C03651=1200.796,212.274,-59.248,-177.519,6.536,148.464
C03652=1200.800,212.025,-59.224,-177.522,6.534,148.465
C03653=1200.805,211.777,-59.199,-177.524,6.533,148.465
C03654=1200.809,211.528,-59.175,-177.527,6.531,148.466
C03655=1200.814,211.257,-59.148,-177.530,6.528,148.466
C03656=1200.819,210.986,-59.122,-177.533,6.526,148.466
C03657=1200.824,210.716,-59.095,-177.535,6.524,148.466
C03658=1200.829,210.446,-59.069,-177.539,6.522,148.467
C03659=1200.833,210.197,-59.044,-177.541,6.520,148.467
C03660=1200.838,209.949,-59.020,-177.543,6.518,148.467
C03661=1200.843,209.700,-58.995,-177.546,6.516,148.468
C03662=1200.847,209.451,-58.971,-177.549,6.514,148.468
C03663=1200.851,209.202,-58.947,-177.551,6.512,148.468
C03664=1200.856,208.953,-58.923,-177.554,6.510,148.469
C03665=1200.861,208.705,-58.899,-177.557,6.509,148.469
C03666=1200.865,208.456,-58.874,-177.559,6.506,148.469
C03667=1200.870,208.207,-58.849,-177.562,6.505,148.469
C03668=1200.874,207.958,-58.825,-177.565,6.502,148.470
C03669=1200.879,207.710,-58.801,-177.567,6.500,148.470
C03670=1200.884,207.461,-58.777,-177.570,6.498,148.470
C03671=1200.888,207.212,-58.753,-177.573,6.497,148.471
C03672=1200.893,206.963,-58.728,-177.575,6.495,148.471
C03673=1200.897,206.714,-58.704,-177.578,6.493,148.471
C03674=1200.902,206.466,-58.680,-177.580,6.491,148.472
C03675=1200.906,206.217,-58.657,-177.583,6.489,148.472
C03676=1200.912,205.968,-58.632,-177.585,6.487,148.472
C03677=1200.915,205.719,-58.608,-177.588,6.485,148.473
C03678=1200.920,205.471,-58.584,-177.591,6.483,148.473
C03679=1200.925,205.221,-58.560,-177.593,6.482,148.473
C03680=1200.930,204.973,-58.536,-177.596,6.480,148.474
C03681=1200.934,204.724,-58.511,-177.598,6.478,148.474
C03682=1200.938,204.475,-58.487,-177.601,6.476,148.474
C03683=1200.943,204.226,-58.463,-177.604,6.474,148.474
C03684=1200.948,203.978,-58.439,-177.606,6.472,148.475
C03685=1200.952,203.729,-58.415,-177.609,6.470,148.475
C03686=1200.957,203.480,-58.392,-177.612,6.468,148.475
C03687=1200.961,203.232,-58.367,-177.615,6.466,148.476
C03688=1200.966,202.982,-58.344,-177.617,6.464,148.476
C03689=1200.970,202.733,-58.319,-177.620,6.462,148.476
C03690=1200.975,202.485,-58.295,-177.622,6.460,148.476
C03691=1200.979,202.236,-58.272,-177.625,6.458,148.477
C03692=1200.984,201.987,-58.248,-177.627,6.456,148.477
C03693=1200.988,201.738,-58.224,-177.630,6.455,148.478
C03694=1200.994,201.490,-58.200,-177.633,6.453,148.478
C03695=1200.998,201.241,-58.176,-177.635,6.451,148.478
C03696=1201.003,200.992,-58.152,-177.638,6.449,148.479
C03697=1201.006,200.743,-58.128,-177.641,6.447,148.479
C03698=1201.011,200.494,-58.104,-177.643,6.446,148.479
C03699=1201.016,200.246,-58.080,-177.646,6.444,148.480
C03700=1201.020,199.997,-58.057,-177.649,6.442,148.480
C03701=1201.025,199.748,-58.033,-177.651,6.440,148.480
C03702=1201.029,199.499,-58.009,-177.654,6.438,148.480
C03703=1201.035,199.250,-57.985,-177.656,6.436,148.481
C03704=1201.039,199.001,-57.961,-177.659,6.434,148.481
C03705=1201.044,198.752,-57.938,-177.661,6.433,148.481
C03706=1201.048,198.504,-57.914,-177.664,6.431,148.482
C03707=1201.053,198.255,-57.891,-177.667,6.429,148.482
C03708=1201.057,198.007,-57.867,-177.669,6.427,148.482
C03709=1201.062,197.758,-57.843,-177.672,6.425,148.483
C03710=1201.067,197.508,-57.820,-177.675,6.423,148.483
C03711=1201.071,197.260,-57.796,-177.677,6.422,148.484
C03712=1201.076,197.011,-57.772,-177.680,6.420,148.484
C03713=1201.080,196.761,-57.749,-177.683,6.418,148.484
C03714=1201.084,196.513,-57.725,-177.685,6.416,148.485
C03715=1201.089,196.264,-57.701,-177.688,6.414,148.485
C03716=1201.094,196.015,-57.678,-177.690,6.412,148.485
C03717=1201.098,195.766,-57.654,-177.693,6.410,148.485
C03718=1201.103,195.517,-57.630,-177.696,6.409,148.486
C03719=1201.108,195.268,-57.607,-177.698,6.407,148.486
C03720=1201.112,195.019,-57.584,-177.701,6.405,148.486
C03721=1201.117,194.771,-57.560,-177.703,6.403,148.487
C03722=1201.121,194.522,-57.536,-177.706,6.401,148.487
C03723=1201.127,194.274,-57.513,-177.709,6.399,148.487
C03724=1201.131,194.025,-57.490,-177.711,6.398,148.488
C03725=1201.136,193.776,-57.466,-177.714,6.396,148.488
C03726=1201.140,193.527,-57.443,-177.717,6.394,148.488
C03727=1201.144,193.278,-57.420,-177.719,6.392,148.489
C03728=1201.149,193.029,-57.396,-177.722,6.390,148.489
C03729=1201.154,192.780,-57.373,-177.725,6.389,148.490
C03730=1201.159,192.531,-57.350,-177.727,6.387,148.490
C03731=1201.163,192.283,-57.326,-177.730,6.385,148.490
C03732=1201.168,192.034,-57.302,-177.733,6.383,148.491
C03733=1201.172,191.785,-57.279,-177.735,6.381,148.491
C03734=1201.177,191.536,-57.256,-177.738,6.380,148.491
C03735=1201.181,191.287,-57.233,-177.741,6.378,148.492
C03736=1201.186,191.038,-57.209,-177.743,6.376,148.492
C03737=1201.190,190.789,-57.186,-177.746,6.374,148.492
C03738=1201.195,190.540,-57.163,-177.748,6.373,148.493
C03739=1201.200,190.292,-57.140,-177.751,6.371,148.493
C03740=1201.205,190.043,-57.116,-177.753,6.369,148.493
C03741=1201.209,189.794,-57.094,-177.756,6.368,148.494
C03742=1201.214,189.545,-57.070,-177.758,6.366,148.494
C03743=1201.218,189.296,-57.047,-177.761,6.364,148.494
C03744=1201.223,189.047,-57.023,-177.764,6.362,148.495
C03745=1201.228,188.798,-57.000,-177.766,6.360,148.495
C03746=1201.232,188.549,-56.977,-177.769,6.358,148.495
C03747=1201.237,188.301,-56.954,-177.772,6.356,148.496
C03748=1201.242,188.052,-56.931,-177.774,6.355,148.496
C03749=1201.247,187.803,-56.908,-177.777,6.353,148.496
C03750=1201.250,187.554,-56.885,-177.779,6.351,148.497
C03751=1201.255,187.305,-56.862,-177.782,6.349,148.497
C03752=1201.260,187.056,-56.838,-177.785,6.347,148.497
C03753=1201.265,186.807,-56.815,-177.787,6.346,148.498
C03754=1201.269,186.559,-56.792,-177.790,6.344,148.498
C03755=1201.274,186.310,-56.769,-177.792,6.343,148.499
C03756=1201.279,186.061,-56.746,-177.795,6.341,148.499
C03757=1201.282,185.812,-56.723,-177.798,6.339,148.499
C03758=1201.288,185.562,-56.700,-177.801,6.338,148.500
C03759=1201.293,185.293,-56.675,-177.803,6.336,148.500
C03760=1201.297,185.024,-56.650,-177.807,6.333,148.500
C03761=1201.302,184.754,-56.625,-177.809,6.331,148.501
C03762=1201.308,184.484,-56.600,-177.812,6.330,148.501
C03763=1201.312,184.235,-56.577,-177.815,6.328,148.502
C03764=1201.317,183.987,-56.555,-177.817,6.326,148.502
C03765=1201.321,183.738,-56.532,-177.820,6.324,148.502
C03766=1201.326,183.489,-56.509,-177.822,6.323,148.503
C03767=1201.331,183.240,-56.486,-177.825,6.321,148.503
C03768=1201.336,182.991,-56.464,-177.827,6.320,148.503
C03769=1201.340,182.742,-56.440,-177.830,6.318,148.504
C03770=1201.344,182.493,-56.418,-177.833,6.316,148.504
C03771=1201.349,182.244,-56.395,-177.836,6.315,148.505
C03772=1201.354,181.995,-56.372,-177.838,6.313,148.505
C03773=1201.358,181.747,-56.349,-177.841,6.311,148.505
C03774=1201.363,181.498,-56.326,-177.844,6.309,148.506
C03775=1201.367,181.248,-56.304,-177.846,6.307,148.506
C03776=1201.372,180.999,-56.281,-177.848,6.306,148.506
C03777=1201.377,180.751,-56.259,-177.851,6.305,148.507
C03778=1201.382,180.502,-56.235,-177.854,6.303,148.507
C03779=1201.386,180.253,-56.213,-177.856,6.301,148.507
C03780=1201.391,180.004,-56.190,-177.859,6.299,148.508
C03781=1201.395,179.755,-56.168,-177.862,6.297,148.508
C03782=1201.400,179.506,-56.144,-177.864,6.296,148.509
C03783=1201.404,179.257,-56.122,-177.867,6.294,148.509
C03784=1201.410,179.008,-56.099,-177.870,6.292,148.509
C03785=1201.414,178.759,-56.077,-177.872,6.291,148.510
C03786=1201.418,178.510,-56.054,-177.875,6.289,148.510
C03787=1201.423,178.261,-56.032,-177.877,6.287,148.510
C03788=1201.428,178.012,-56.009,-177.880,6.286,148.511
C03789=1201.432,177.763,-55.987,-177.883,6.284,148.511
C03790=1201.438,177.515,-55.964,-177.886,6.282,148.512
C03791=1201.442,177.265,-55.942,-177.888,6.280,148.512
C03792=1201.447,177.016,-55.918,-177.890,6.279,148.512
C03793=1201.451,176.768,-55.897,-177.893,6.278,148.513
C03794=1201.455,176.519,-55.874,-177.896,6.276,148.513
C03795=1201.460,176.269,-55.851,-177.898,6.274,148.514
C03796=1201.465,176.021,-55.829,-177.901,6.272,148.514
C03797=1201.470,175.772,-55.806,-177.904,6.270,148.514
C03798=1201.474,175.522,-55.784,-177.906,6.269,148.515
C03799=1201.479,175.274,-55.762,-177.909,6.268,148.515
C03800=1201.484,175.025,-55.739,-177.911,6.266,148.515
C03801=1201.488,174.777,-55.717,-177.914,6.264,148.516
C03802=1201.493,174.527,-55.695,-177.917,6.262,148.516
C03803=1201.498,174.278,-55.672,-177.920,6.261,148.517
C03804=1201.502,174.030,-55.650,-177.922,6.259,148.517
C03805=1201.506,173.780,-55.628,-177.925,6.257,148.517
C03806=1201.512,173.531,-55.605,-177.927,6.256,148.518
C03807=1201.516,173.283,-55.583,-177.930,6.254,148.518
C03808=1201.520,173.033,-55.561,-177.932,6.253,148.518
C03809=1201.526,172.784,-55.538,-177.935,6.251,148.519
C03810=1201.530,172.536,-55.515,-177.938,6.249,148.519
C03811=1201.535,172.287,-55.494,-177.940,6.247,148.520
C03812=1201.540,172.037,-55.471,-177.943,6.246,148.520
C03813=1201.545,171.789,-55.449,-177.946,6.245,148.521
C03814=1201.549,171.540,-55.427,-177.948,6.243,148.521
C03815=1201.554,171.290,-55.404,-177.951,6.241,148.521
C03816=1201.558,171.042,-55.382,-177.954,6.239,148.522
C03817=1201.563,170.792,-55.360,-177.956,6.238,148.522
C03818=1201.567,170.544,-55.338,-177.958,6.237,148.522
C03819=1201.572,170.295,-55.315,-177.961,6.235,148.523
C03820=1201.577,170.046,-55.294,-177.964,6.233,148.523
C03821=1201.581,169.797,-55.272,-177.966,6.231,148.523
C03822=1201.586,169.548,-55.250,-177.970,6.230,148.524
C03823=1201.591,169.299,-55.228,-177.972,6.229,148.524
C03824=1201.596,169.050,-55.205,-177.974,6.227,148.525
C03825=1201.600,168.801,-55.183,-177.977,6.225,148.525
C03826=1201.605,168.552,-55.161,-177.980,6.223,148.526
C03827=1201.609,168.303,-55.139,-177.982,6.222,148.526
C03828=1201.614,168.054,-55.117,-177.985,6.221,148.526
C03829=1201.619,167.805,-55.095,-177.987,6.219,148.527
C03830=1201.624,167.556,-55.073,-177.990,6.217,148.527
C03831=1201.628,167.307,-55.051,-177.993,6.216,148.528
C03832=1201.633,167.058,-55.029,-177.996,6.214,148.528
C03833=1201.637,166.809,-55.007,-177.998,6.213,148.528
C03834=1201.642,166.560,-54.986,-178.000,6.211,148.529
C03835=1201.647,166.311,-54.964,-178.003,6.209,148.529
C03836=1201.652,166.062,-54.941,-178.006,6.207,148.529
C03837=1201.656,165.812,-54.919,-178.009,6.206,148.530
C03838=1201.661,165.564,-54.898,-178.011,6.205,148.530
C03839=1201.666,165.315,-54.876,-178.014,6.203,148.531
C03840=1201.670,165.066,-54.854,-178.016,6.201,148.531
C03841=1201.675,164.817,-54.832,-178.019,6.200,148.532
C03842=1201.680,164.568,-54.810,-178.022,6.198,148.532
C03843=1201.684,164.319,-54.788,-178.024,6.197,148.532
C03844=1201.689,164.070,-54.766,-178.027,6.195,148.533
C03845=1201.694,163.821,-54.745,-178.030,6.194,148.533
C03846=1201.698,163.572,-54.723,-178.032,6.192,148.534
C03847=1201.703,163.323,-54.701,-178.034,6.191,148.534
C03848=1201.708,163.075,-54.679,-178.037,6.189,148.534
C03849=1201.712,162.825,-54.657,-178.040,6.187,148.535
C03850=1201.717,162.577,-54.636,-178.043,6.186,148.535
C03851=1201.721,162.327,-54.614,-178.045,6.185,148.536
C03852=1201.726,162.078,-54.593,-178.048,6.183,148.536
C03853=1201.731,161.829,-54.571,-178.050,6.181,148.536
C03854=1201.735,161.580,-54.549,-178.053,6.179,148.537
C03855=1201.740,161.331,-54.527,-178.056,6.178,148.537
C03856=1201.744,161.082,-54.505,-178.058,6.177,148.538
C03857=1201.750,160.833,-54.484,-178.061,6.175,148.538
C03858=1201.755,160.584,-54.462,-178.064,6.173,148.539
C03859=1201.759,160.335,-54.440,-178.066,6.172,148.539
C03860=1201.764,160.086,-54.419,-178.068,6.171,148.539
C03861=1201.769,159.837,-54.398,-178.071,6.169,148.540
C03862=1201.773,159.588,-54.376,-178.074,6.167,148.540
C03863=1201.779,159.318,-54.352,-178.077,6.166,148.541
C03864=1201.783,159.050,-54.329,-178.080,6.164,148.541
C03865=1201.788,158.780,-54.305,-178.083,6.162,148.542
C03866=1201.793,158.511,-54.283,-178.085,6.161,148.542
C03867=1201.798,158.263,-54.261,-178.088,6.160,148.542
C03868=1201.803,158.014,-54.239,-178.091,6.158,148.543
C03869=1201.808,157.764,-54.218,-178.093,6.156,148.543
C03870=1201.812,157.516,-54.196,-178.096,6.155,148.544
C03871=1201.817,157.267,-54.175,-178.098,6.154,148.544
C03872=1201.821,157.017,-54.154,-178.101,6.152,148.544
C03873=1201.826,156.769,-54.132,-178.104,6.150,148.545
C03874=1201.831,156.520,-54.111,-178.107,6.149,148.545
C03875=1201.836,156.271,-54.090,-178.109,6.148,148.546
C03876=1201.840,156.021,-54.068,-178.111,6.146,148.546
C03877=1201.845,155.772,-54.047,-178.114,6.144,148.547
C03878=1201.850,155.524,-54.025,-178.117,6.143,148.547
C03879=1201.855,155.275,-54.005,-178.119,6.142,148.548
C03880=1201.859,155.025,-53.982,-178.122,6.140,148.548
C03881=1201.864,154.777,-53.961,-178.125,6.138,148.548
C03882=1201.869,154.527,-53.940,-178.127,6.137,148.549
C03883=1201.873,154.278,-53.918,-178.130,6.136,148.549
C03884=1201.878,154.029,-53.897,-178.133,6.134,148.550
C03885=1201.883,153.780,-53.876,-178.135,6.133,148.550
C03886=1201.888,153.531,-53.855,-178.137,6.131,148.550
C03887=1201.893,153.282,-53.833,-178.140,6.129,148.551
C03888=1201.897,153.033,-53.812,-178.143,6.128,148.551
C03889=1201.902,152.784,-53.791,-178.145,6.127,148.552
C03890=1201.907,152.535,-53.770,-178.148,6.125,148.552
C03891=1201.911,152.286,-53.749,-178.151,6.123,148.553
C03892=1201.915,152.037,-53.727,-178.153,6.123,148.553
C03893=1201.920,151.787,-53.706,-178.156,6.121,148.554
C03894=1201.925,151.539,-53.685,-178.159,6.119,148.554
C03895=1201.930,151.290,-53.664,-178.161,6.118,148.554
C03896=1201.935,151.041,-53.643,-178.164,6.117,148.555
C03897=1201.939,150.791,-53.621,-178.167,6.115,148.555
C03898=1201.944,150.542,-53.601,-178.169,6.113,148.556
C03899=1201.949,150.293,-53.580,-178.171,6.112,148.556
C03900=1201.954,150.044,-53.558,-178.175,6.111,148.557
C03901=1201.958,149.795,-53.538,-178.177,6.109,148.557
C03902=1201.963,149.546,-53.517,-178.179,6.108,148.557
C03903=1201.968,149.297,-53.495,-178.182,6.106,148.558
C03904=1201.972,149.048,-53.474,-178.185,6.105,148.558
C03905=1201.977,148.799,-53.453,-178.187,6.104,148.559
C03906=1201.982,148.550,-53.432,-178.190,6.102,148.559
C03907=1201.987,148.301,-53.411,-178.193,6.100,148.560
C03908=1201.992,148.052,-53.390,-178.195,6.100,148.560
C03909=1201.996,147.803,-53.370,-178.198,6.098,148.561
C03910=1202.000,147.553,-53.348,-178.201,6.096,148.561
C03911=1202.006,147.304,-53.327,-178.203,6.095,148.561
C03912=1202.010,147.055,-53.307,-178.206,6.094,148.562
C03913=1202.015,146.806,-53.286,-178.209,6.092,148.562
C03914=1202.019,146.558,-53.265,-178.211,6.091,148.563
C03915=1202.024,146.308,-53.244,-178.213,6.089,148.563
C03916=1202.029,146.059,-53.223,-178.217,6.088,148.564
C03917=1202.034,145.810,-53.202,-178.219,6.087,148.564
C03918=1202.039,145.560,-53.181,-178.221,6.085,148.565
C03919=1202.043,145.311,-53.161,-178.224,6.083,148.565
C03920=1202.048,145.063,-53.139,-178.227,6.082,148.566
C03921=1202.052,144.814,-53.119,-178.229,6.081,148.566
C03922=1202.058,144.564,-53.098,-178.232,6.079,148.566
C03923=1202.062,144.315,-53.077,-178.235,6.078,148.567
C03924=1202.067,144.066,-53.056,-178.237,6.076,148.567
C03925=1202.072,143.817,-53.036,-178.240,6.075,148.568
C03926=1202.077,143.568,-53.015,-178.242,6.074,148.568
C03927=1202.081,143.319,-52.995,-178.245,6.072,148.569
C03928=1202.086,143.070,-52.974,-178.247,6.071,148.569
C03929=1202.091,142.821,-52.953,-178.250,6.070,148.569
C03930=1202.095,142.572,-52.933,-178.253,6.068,148.570
C03931=1202.100,142.323,-52.912,-178.255,6.067,148.570
C03932=1202.105,142.074,-52.891,-178.258,6.065,148.571
C03933=1202.109,141.824,-52.869,-178.261,6.064,148.571
C03934=1202.114,141.575,-52.849,-178.263,6.063,148.572
C03935=1202.119,141.326,-52.828,-178.266,6.061,148.572
C03936=1202.124,141.077,-52.808,-178.269,6.059,148.573
C03937=1202.128,140.828,-52.788,-178.271,6.059,148.573
C03938=1202.133,140.578,-52.767,-178.274,6.057,148.574
C03939=1202.138,140.329,-52.747,-178.276,6.056,148.574
C03940=1202.143,140.080,-52.726,-178.279,6.055,148.575
C03941=1202.147,139.831,-52.705,-178.282,6.053,148.575
C03942=1202.152,139.582,-52.685,-178.284,6.052,148.575
C03943=1202.157,139.333,-52.664,-178.287,6.050,148.576
C03944=1202.161,139.084,-52.644,-178.289,6.050,148.576
C03945=1202.166,138.835,-52.623,-178.292,6.048,148.577
C03946=1202.171,138.586,-52.602,-178.295,6.046,148.577
C03947=1202.175,138.337,-52.582,-178.297,6.045,148.578
C03948=1202.180,138.087,-52.562,-178.300,6.044,148.578
C03949=1202.186,137.839,-52.542,-178.303,6.042,148.579
C03950=1202.190,137.590,-52.521,-178.305,6.041,148.579
C03951=1202.195,137.341,-52.501,-178.308,6.039,148.580
C03952=1202.200,137.092,-52.480,-178.310,6.038,148.580
C03953=1202.204,136.843,-52.460,-178.313,6.037,148.581
C03954=1202.209,136.593,-52.440,-178.316,6.035,148.581
C03955=1202.214,136.344,-52.419,-178.318,6.034,148.581
C03956=1202.219,136.095,-52.399,-178.321,6.033,148.582
C03957=1202.223,135.846,-52.378,-178.323,6.032,148.582
C03958=1202.228,135.596,-52.359,-178.326,6.030,148.583
C03959=1202.233,135.347,-52.338,-178.329,6.029,148.583
C03960=1202.237,135.098,-52.317,-178.331,6.028,148.584
C03961=1202.242,134.849,-52.297,-178.334,6.026,148.584
C03962=1202.247,134.600,-52.277,-178.337,6.025,148.585
C03963=1202.252,134.351,-52.257,-178.339,6.024,148.585
C03964=1202.257,134.102,-52.236,-178.341,6.023,148.586
C03965=1202.261,133.853,-52.216,-178.344,6.021,148.586
C03966=1202.266,133.604,-52.196,-178.347,6.019,148.587
C03967=1202.271,133.335,-52.174,-178.350,6.019,148.587
C03968=1202.276,133.067,-52.153,-178.352,6.017,148.588
C03969=1202.282,132.798,-52.130,-178.356,6.016,148.588
C03970=1202.287,132.529,-52.108,-178.358,6.014,148.589
C03971=1202.292,132.280,-52.088,-178.361,6.013,148.589
C03972=1202.296,132.031,-52.069,-178.364,6.011,148.590
C03973=1202.301,131.782,-52.048,-178.366,6.010,148.590
C03974=1202.306,131.532,-52.029,-178.369,6.009,148.591
C03975=1202.310,131.283,-52.008,-178.372,6.007,148.591
C03976=1202.315,131.034,-51.988,-178.374,6.006,148.592
C03977=1202.320,130.784,-51.968,-178.377,6.005,148.592
C03978=1202.325,130.536,-51.948,-178.379,6.004,148.593
C03979=1202.330,130.287,-51.928,-178.382,6.002,148.593
C03980=1202.334,130.038,-51.908,-178.384,6.002,148.594
C03981=1202.339,129.788,-51.888,-178.387,6.000,148.594
C03982=1202.343,129.539,-51.868,-178.390,5.999,148.595
C03983=1202.349,129.290,-51.848,-178.392,5.997,148.595
C03984=1202.353,129.041,-51.828,-178.395,5.996,148.595
C03985=1202.358,128.792,-51.808,-178.398,5.995,148.596
C03986=1202.363,128.543,-51.787,-178.400,5.993,148.596
C03987=1202.368,128.293,-51.768,-178.402,5.992,148.597
C03988=1202.373,128.045,-51.748,-178.406,5.991,148.597
C03989=1202.378,127.795,-51.728,-178.408,5.990,148.598
C03990=1202.382,127.546,-51.708,-178.411,5.989,148.598
C03991=1202.387,127.297,-51.688,-178.413,5.988,148.599
C03992=1202.392,127.047,-51.668,-178.416,5.986,148.599
C03993=1202.397,126.799,-51.648,-178.418,5.985,148.600
C03994=1202.401,126.549,-51.629,-178.421,5.983,148.600
C03995=1202.406,126.300,-51.608,-178.424,5.982,148.601
C03996=1202.410,126.051,-51.589,-178.426,5.981,148.601
C03997=1202.416,125.802,-51.569,-178.429,5.979,148.602
C03998=1202.420,125.553,-51.549,-178.432,5.979,148.602
C03999=1202.425,125.303,-51.529,-178.434,5.977,148.603
C04000=1202.430,125.054,-51.510,-178.436,5.976,148.603
C04001=1202.435,124.806,-51.490,-178.440,5.975,148.604
C04002=1202.440,124.556,-51.470,-178.442,5.974,148.604
C04003=1202.444,124.306,-51.450,-178.445,5.972,148.605
C04004=1202.449,124.057,-51.430,-178.447,5.971,148.605
C04005=1202.454,123.809,-51.411,-178.450,5.969,148.606
C04006=1202.458,123.559,-51.392,-178.452,5.969,148.606
C04007=1202.463,123.310,-51.372,-178.455,5.967,148.607
C04008=1202.468,123.062,-51.352,-178.458,5.967,148.607
C04009=1202.473,122.812,-51.332,-178.460,5.965,148.608
C04010=1202.477,122.562,-51.313,-178.462,5.964,148.608
C04011=1202.482,122.313,-51.293,-178.466,5.962,148.609
C04012=1202.487,122.065,-51.273,-178.468,5.961,148.609
C04013=1202.492,121.815,-51.253,-178.471,5.960,148.610
C04014=1202.497,121.565,-51.234,-178.473,5.959,148.610
C04015=1202.502,121.317,-51.214,-178.476,5.957,148.610
C04016=1202.506,121.067,-51.195,-178.478,5.957,148.611
C04017=1202.510,120.818,-51.175,-178.481,5.955,148.611
C04018=1202.516,120.570,-51.156,-178.484,5.954,148.612
C04019=1202.520,120.320,-51.136,-178.486,5.953,148.613
C04020=1202.525,120.070,-51.116,-178.489,5.952,148.613
C04021=1202.531,119.821,-51.097,-178.492,5.950,148.614
C04022=1202.535,119.572,-51.077,-178.494,5.949,148.614
C04023=1202.539,119.323,-51.058,-178.497,5.948,148.615
C04024=1202.544,119.074,-51.038,-178.499,5.947,148.615
C04025=1202.549,118.825,-51.019,-178.502,5.945,148.616
C04026=1202.554,118.576,-50.999,-178.504,5.945,148.616
C04027=1202.559,118.326,-50.980,-178.507,5.943,148.617
C04028=1202.563,118.077,-50.961,-178.510,5.942,148.617
C04029=1202.569,117.828,-50.941,-178.512,5.940,148.617
C04030=1202.573,117.579,-50.922,-178.515,5.940,148.618
C04031=1202.578,117.329,-50.902,-178.518,5.938,148.619
C04032=1202.583,117.081,-50.883,-178.520,5.937,148.619
C04033=1202.587,116.831,-50.864,-178.523,5.936,148.620
C04034=1202.593,116.582,-50.844,-178.525,5.935,148.620
C04035=1202.597,116.333,-50.825,-178.528,5.933,148.621
C04036=1202.602,116.084,-50.806,-178.531,5.933,148.621
C04037=1202.607,115.834,-50.786,-178.533,5.931,148.622
C04038=1202.612,115.585,-50.767,-178.536,5.930,148.622
C04039=1202.617,115.336,-50.747,-178.538,5.929,148.623
C04040=1202.621,115.087,-50.728,-178.541,5.928,148.623
C04041=1202.626,114.838,-50.709,-178.544,5.927,148.624
C04042=1202.631,114.588,-50.689,-178.546,5.925,148.624
C04043=1202.636,114.340,-50.671,-178.549,5.925,148.625
C04044=1202.640,114.090,-50.651,-178.552,5.923,148.625
C04045=1202.645,113.840,-50.632,-178.554,5.922,148.626
C04046=1202.651,113.591,-50.613,-178.557,5.921,148.626
C04047=1202.655,113.342,-50.594,-178.559,5.920,148.627
C04048=1202.660,113.093,-50.574,-178.562,5.918,148.627
C04049=1202.665,112.843,-50.555,-178.564,5.917,148.628
C04050=1202.669,112.595,-50.536,-178.567,5.917,148.628
C04051=1202.674,112.345,-50.516,-178.570,5.915,148.629
C04052=1202.679,112.096,-50.498,-178.572,5.914,148.629
C04053=1202.684,111.847,-50.479,-178.575,5.913,148.630
C04054=1202.689,111.598,-50.460,-178.577,5.912,148.630
C04055=1202.693,111.348,-50.440,-178.580,5.910,148.631
C04056=1202.699,111.100,-50.421,-178.583,5.910,148.631
C04057=1202.703,110.850,-50.402,-178.586,5.908,148.632
C04058=1202.708,110.601,-50.384,-178.588,5.907,148.632
C04059=1202.713,110.351,-50.364,-178.590,5.906,148.633
C04060=1202.718,110.103,-50.345,-178.593,5.905,148.633
C04061=1202.722,109.853,-50.326,-178.596,5.904,148.634
C04062=1202.727,109.604,-50.308,-178.599,5.903,148.635
C04063=1202.732,109.354,-50.288,-178.601,5.902,148.635
C04064=1202.737,109.106,-50.269,-178.604,5.900,148.635
C04065=1202.742,108.856,-50.250,-178.606,5.899,148.636
C04066=1202.747,108.607,-50.231,-178.608,5.898,148.636
C04067=1202.751,108.358,-50.212,-178.611,5.897,148.637
C04068=1202.757,108.108,-50.193,-178.614,5.896,148.637
C04069=1202.761,107.860,-50.175,-178.617,5.895,148.638
C04070=1202.766,107.610,-50.155,-178.619,5.894,148.638
C04071=1202.771,107.342,-50.136,-178.622,5.892,148.639
C04072=1202.776,107.073,-50.115,-178.625,5.892,148.640
C04073=1202.782,106.804,-50.095,-178.627,5.890,148.640
C04074=1202.787,106.537,-50.074,-178.631,5.889,148.641
C04075=1202.791,106.287,-50.055,-178.633,5.888,148.641
C04076=1202.796,106.038,-50.037,-178.635,5.887,148.642
C04077=1202.801,105.789,-50.017,-178.639,5.886,148.642
C04078=1202.806,105.539,-49.999,-178.641,5.885,148.643
C04079=1202.811,105.290,-49.979,-178.644,5.883,148.644
C04080=1202.815,105.041,-49.961,-178.646,5.882,148.644
C04081=1202.821,104.792,-49.942,-178.649,5.882,148.645
C04082=1202.825,104.542,-49.923,-178.651,5.880,148.645
C04083=1202.830,104.293,-49.905,-178.654,5.879,148.646
C04084=1202.835,104.044,-49.886,-178.657,5.878,148.646
C04085=1202.839,103.795,-49.868,-178.659,5.877,148.647
C04086=1202.845,103.546,-49.848,-178.661,5.876,148.647
C04087=1202.849,103.296,-49.830,-178.665,5.875,148.648
C04088=1202.854,103.047,-49.811,-178.667,5.874,148.648
C04089=1202.859,102.798,-49.793,-178.670,5.872,148.649
C04090=1202.863,102.549,-49.774,-178.672,5.871,148.649
C04091=1202.869,102.299,-49.755,-178.675,5.871,148.650
C04092=1202.874,102.050,-49.737,-178.677,5.869,148.650
C04093=1202.878,101.801,-49.718,-178.680,5.869,148.651
C04094=1202.884,101.551,-49.699,-178.682,5.868,148.651
C04095=1202.888,101.303,-49.681,-178.685,5.866,148.652
C04096=1202.892,101.053,-49.662,-178.687,5.865,148.652
C04097=1202.898,100.804,-49.643,-178.691,5.864,148.653
C04098=1202.903,100.555,-49.625,-178.693,5.863,148.653
C04099=1202.907,100.305,-49.607,-178.695,5.862,148.654
C04100=1202.912,100.056,-49.587,-178.698,5.861,148.654
C04101=1202.917,99.807,-49.569,-178.701,5.860,148.655
C04102=1202.922,99.557,-49.551,-178.703,5.859,148.656
C04103=1202.927,99.308,-49.532,-178.706,5.858,148.656
C04104=1202.932,99.059,-49.514,-178.709,5.857,148.657
C04105=1202.936,98.809,-49.495,-178.711,5.855,148.657
C04106=1202.941,98.560,-49.477,-178.714,5.855,148.658
C04107=1202.946,98.311,-49.458,-178.716,5.854,148.658
C04108=1202.951,98.062,-49.440,-178.719,5.852,148.659
C04109=1202.955,97.812,-49.421,-178.721,5.852,148.659
C04110=1202.960,97.563,-49.403,-178.724,5.851,148.660
C04111=1202.966,97.314,-49.385,-178.727,5.849,148.660
C04112=1202.971,97.065,-49.367,-178.729,5.849,148.661
C04113=1202.975,96.815,-49.348,-178.731,5.848,148.662
C04114=1202.980,96.566,-49.330,-178.735,5.846,148.662
C04115=1202.985,96.317,-49.311,-178.737,5.845,148.663
C04116=1202.990,96.068,-49.293,-178.739,5.845,148.663
C04117=1202.994,95.818,-49.274,-178.743,5.843,148.664
C04118=1202.999,95.569,-49.256,-178.745,5.842,148.664
C04119=1203.004,95.320,-49.238,-178.748,5.841,148.665
C04120=1203.010,95.070,-49.219,-178.750,5.840,148.665
C04121=1203.014,94.821,-49.201,-178.753,5.840,148.666
C04122=1203.019,94.571,-49.183,-178.755,5.838,148.666
C04123=1203.024,94.323,-49.164,-178.758,5.837,148.667
C04124=1203.028,94.074,-49.146,-178.760,5.836,148.667
C04125=1203.033,93.824,-49.128,-178.763,5.835,148.668
C04126=1203.038,93.574,-49.109,-178.766,5.834,148.669
C04127=1203.043,93.325,-49.092,-178.768,5.833,148.669
C04128=1203.048,93.076,-49.074,-178.771,5.832,148.670
C04129=1203.053,92.827,-49.056,-178.773,5.831,148.670
C04130=1203.058,92.577,-49.037,-178.776,5.831,148.671
C04131=1203.062,92.328,-49.019,-178.779,5.829,148.671
C04132=1203.067,92.079,-49.001,-178.781,5.828,148.672
C04133=1203.072,91.830,-48.983,-178.784,5.828,148.673
C04134=1203.077,91.581,-48.965,-178.787,5.826,148.673
C04135=1203.082,91.332,-48.947,-178.789,5.825,148.674
C04136=1203.087,91.081,-48.928,-178.791,5.824,148.674
C04137=1203.092,90.832,-48.910,-178.794,5.824,148.675
C04138=1203.097,90.583,-48.892,-178.797,5.822,148.675
C04139=1203.102,90.334,-48.874,-178.799,5.822,148.676
C04140=1203.106,90.085,-48.856,-178.802,5.821,148.676
C04141=1203.111,89.836,-48.838,-178.805,5.819,148.677
C04142=1203.116,89.586,-48.819,-178.807,5.819,148.678
C04143=1203.121,89.336,-48.801,-178.809,5.818,148.678
C04144=1203.125,89.087,-48.783,-178.813,5.816,148.679
C04145=1203.130,88.838,-48.765,-178.815,5.815,148.679
C04146=1203.135,88.589,-48.747,-178.817,5.815,148.680
C04147=1203.140,88.340,-48.730,-178.821,5.813,148.680
C04148=1203.145,88.090,-48.712,-178.823,5.812,148.681
C04149=1203.150,87.841,-48.694,-178.825,5.812,148.681
C04150=1203.155,87.592,-48.676,-178.827,5.811,148.682
C04151=1203.160,87.342,-48.658,-178.831,5.810,148.682
C04152=1203.164,87.093,-48.640,-178.833,5.809,148.683
C04153=1203.169,86.843,-48.622,-178.835,5.808,148.684
C04154=1203.174,86.594,-48.604,-178.839,5.807,148.684
C04155=1203.179,86.345,-48.586,-178.841,5.806,148.685
C04156=1203.184,86.095,-48.569,-178.843,5.805,148.685
C04157=1203.189,85.846,-48.551,-178.847,5.804,148.686
C04158=1203.194,85.597,-48.533,-178.849,5.803,148.686
C04159=1203.199,85.348,-48.515,-178.851,5.802,148.687
C04160=1203.204,85.099,-48.497,-178.853,5.801,148.687
C04161=1203.208,84.850,-48.479,-178.857,5.800,148.688
C04162=1203.213,84.600,-48.462,-178.859,5.799,148.689
C04163=1203.218,84.350,-48.444,-178.861,5.799,148.689
C04164=1203.223,84.101,-48.426,-178.865,5.797,148.690
C04165=1203.228,83.852,-48.408,-178.867,5.796,148.690
C04166=1203.233,83.602,-48.391,-178.869,5.796,148.691
C04167=1203.238,83.353,-48.373,-178.872,5.795,148.692
C04168=1203.243,83.104,-48.355,-178.875,5.793,148.692
C04169=1203.248,82.854,-48.337,-178.877,5.793,148.693
C04170=1203.252,82.605,-48.320,-178.879,5.792,148.693
C04171=1203.257,82.356,-48.302,-178.882,5.791,148.694
C04172=1203.262,82.107,-48.284,-178.885,5.790,148.694
C04173=1203.267,81.857,-48.266,-178.887,5.789,148.695
C04174=1203.272,81.608,-48.249,-178.890,5.788,148.695
C04175=1203.277,81.339,-48.229,-178.893,5.787,148.696
C04176=1203.282,81.070,-48.211,-178.895,5.786,148.696
C04177=1203.288,80.803,-48.192,-178.899,5.785,148.697
C04178=1203.294,80.534,-48.173,-178.901,5.784,148.698
C04179=1203.298,80.285,-48.156,-178.904,5.784,148.698
C04180=1203.303,80.036,-48.138,-178.906,5.783,148.699
C04181=1203.308,79.786,-48.120,-178.909,5.781,148.699
C04182=1203.313,79.537,-48.102,-178.912,5.781,148.700
C04183=1203.317,79.288,-48.086,-178.914,5.780,148.701
C04184=1203.322,79.038,-48.068,-178.917,5.778,148.701
C04185=1203.327,78.789,-48.050,-178.919,5.778,148.702
C04186=1203.332,78.539,-48.032,-178.922,5.777,148.702
C04187=1203.337,78.290,-48.014,-178.925,5.776,148.703
C04188=1203.342,78.041,-47.998,-178.927,5.775,148.703
C04189=1203.347,77.792,-47.980,-178.930,5.774,148.704
C04190=1203.352,77.542,-47.963,-178.933,5.774,148.705
C04191=1203.357,77.293,-47.945,-178.935,5.773,148.705
C04192=1203.361,77.043,-47.928,-178.937,5.772,148.706
C04193=1203.366,76.794,-47.910,-178.940,5.771,148.706
C04194=1203.372,76.545,-47.893,-178.943,5.770,148.707
C04195=1203.376,76.296,-47.876,-178.945,5.769,148.708
C04196=1203.381,76.046,-47.858,-178.947,5.768,148.708
C04197=1203.386,75.797,-47.840,-178.951,5.767,148.709
C04198=1203.391,75.547,-47.824,-178.953,5.766,148.709
C04199=1203.396,75.298,-47.806,-178.955,5.765,148.710
C04200=1203.401,75.049,-47.789,-178.958,5.765,148.710
C04201=1203.405,74.800,-47.771,-178.961,5.764,148.711
C04202=1203.410,74.550,-47.754,-178.963,5.763,148.711
C04203=1203.415,74.301,-47.736,-178.966,5.762,148.712
C04204=1203.420,74.051,-47.719,-178.969,5.761,148.713
C04205=1203.425,73.802,-47.702,-178.971,5.761,148.713
C04206=1203.430,73.553,-47.684,-178.974,5.759,148.714
C04207=1203.435,73.303,-47.668,-178.977,5.759,148.714
C04208=1203.440,73.054,-47.650,-178.979,5.758,148.715
C04209=1203.445,72.804,-47.632,-178.981,5.757,148.716
C04210=1203.449,72.555,-47.616,-178.984,5.755,148.716
C04211=1203.454,72.306,-47.598,-178.987,5.755,148.717
C04212=1203.459,72.057,-47.581,-178.989,5.754,148.717
C04213=1203.465,71.807,-47.564,-178.991,5.753,148.718
C04214=1203.469,71.558,-47.547,-178.994,5.753,148.718
C04215=1203.474,71.309,-47.530,-178.997,5.751,148.719
C04216=1203.479,71.059,-47.512,-178.999,5.751,148.719
C04217=1203.484,70.809,-47.496,-179.002,5.750,148.720
C04218=1203.489,70.561,-47.478,-179.005,5.749,148.721
C04219=1203.494,70.311,-47.461,-179.007,5.749,148.721
C04220=1203.499,70.062,-47.444,-179.010,5.747,148.722
C04221=1203.503,69.812,-47.427,-179.013,5.747,148.723
C04222=1203.508,69.563,-47.409,-179.015,5.746,148.723
C04223=1203.513,69.313,-47.393,-179.017,5.745,148.724
C04224=1203.519,69.064,-47.376,-179.020,5.745,148.724
C04225=1203.523,68.815,-47.359,-179.023,5.743,148.725
C04226=1203.528,68.566,-47.341,-179.025,5.742,148.725
C04227=1203.533,68.316,-47.325,-179.028,5.742,148.726
C04228=1203.538,68.066,-47.307,-179.030,5.741,148.726
C04229=1203.543,67.818,-47.291,-179.033,5.740,148.727
C04230=1203.548,67.568,-47.274,-179.035,5.740,148.728
C04231=1203.552,67.319,-47.256,-179.038,5.738,148.728
C04232=1203.557,67.069,-47.239,-179.041,5.737,148.729
C04233=1203.563,66.820,-47.223,-179.043,5.737,148.730
C04234=1203.568,66.571,-47.205,-179.046,5.736,148.730
C04235=1203.572,66.321,-47.189,-179.048,5.735,148.731
C04236=1203.577,66.071,-47.172,-179.051,5.734,148.731
C04237=1203.582,65.822,-47.155,-179.054,5.733,148.732
C04238=1203.588,65.573,-47.138,-179.056,5.733,148.732
C04239=1203.592,65.324,-47.121,-179.059,5.732,148.733
C04240=1203.596,65.074,-47.104,-179.061,5.731,148.734
C04241=1203.602,64.825,-47.087,-179.064,5.731,148.734
C04242=1203.607,64.576,-47.070,-179.067,5.729,148.735
C04243=1203.612,64.326,-47.053,-179.069,5.729,148.735
C04244=1203.616,64.076,-47.036,-179.072,5.728,148.736
C04245=1203.621,63.828,-47.020,-179.074,5.727,148.737
C04246=1203.627,63.578,-47.003,-179.077,5.727,148.737
C04247=1203.631,63.328,-46.986,-179.079,5.726,148.738
C04248=1203.636,63.079,-46.969,-179.082,5.724,148.738
C04249=1203.641,62.830,-46.953,-179.085,5.724,148.739
C04250=1203.646,62.580,-46.936,-179.087,5.723,148.739
C04251=1203.651,62.331,-46.919,-179.090,5.722,148.740
C04252=1203.656,62.082,-46.902,-179.092,5.722,148.741
C04253=1203.661,61.832,-46.886,-179.095,5.721,148.741
C04254=1203.666,61.582,-46.868,-179.098,5.720,148.742
C04255=1203.671,61.334,-46.852,-179.100,5.719,148.743
C04256=1203.676,61.084,-46.835,-179.103,5.718,148.743
C04257=1203.681,60.834,-46.818,-179.105,5.718,148.744
C04258=1203.686,60.586,-46.802,-179.108,5.717,148.744
C04259=1203.690,60.336,-46.785,-179.110,5.716,148.745
C04260=1203.696,60.086,-46.769,-179.112,5.715,148.745
C04261=1203.701,59.837,-46.752,-179.116,5.714,148.746
C04262=1203.705,59.587,-46.736,-179.118,5.714,148.747
C04263=1203.710,59.338,-46.719,-179.121,5.713,148.747
C04264=1203.716,59.089,-46.702,-179.123,5.712,148.748
C04265=1203.720,58.839,-46.685,-179.126,5.712,148.748
C04266=1203.725,58.590,-46.669,-179.128,5.711,148.749
C04267=1203.730,58.341,-46.653,-179.130,5.710,148.750
C04268=1203.735,58.091,-46.636,-179.134,5.709,148.750
C04269=1203.740,57.842,-46.620,-179.136,5.708,148.751
C04270=1203.745,57.592,-46.603,-179.139,5.708,148.752
C04271=1203.749,57.343,-46.586,-179.141,5.707,148.752
C04272=1203.755,57.094,-46.569,-179.144,5.706,148.753
C04273=1203.760,56.844,-46.553,-179.146,5.706,148.753
C04274=1203.764,56.594,-46.537,-179.148,5.705,148.754
C04275=1203.769,56.346,-46.520,-179.151,5.704,148.754
C04276=1203.775,56.096,-46.503,-179.154,5.703,148.755
C04277=1203.780,55.847,-46.487,-179.157,5.702,148.756
C04278=1203.785,55.597,-46.471,-179.159,5.701,148.756
C04279=1203.790,55.329,-46.453,-179.162,5.701,148.757
C04280=1203.795,55.060,-46.436,-179.164,5.700,148.758
C04281=1203.801,54.792,-46.418,-179.168,5.699,148.758
C04282=1203.806,54.523,-46.401,-179.170,5.698,148.759
C04283=1203.811,54.274,-46.384,-179.173,5.698,148.760
C04284=1203.815,54.024,-46.367,-179.175,5.697,148.760
C04285=1203.820,53.775,-46.351,-179.178,5.696,148.761
C04286=1203.825,53.525,-46.335,-179.180,5.696,148.761
C04287=1203.831,53.276,-46.318,-179.183,5.695,148.762
C04288=1203.835,53.027,-46.301,-179.186,5.694,148.762
C04289=1203.841,52.777,-46.286,-179.188,5.693,148.763
C04290=1203.845,52.528,-46.269,-179.191,5.693,148.764
C04291=1203.851,52.278,-46.254,-179.194,5.692,148.764
C04292=1203.855,52.029,-46.237,-179.196,5.691,148.765
C04293=1203.860,51.780,-46.221,-179.198,5.691,148.766
C04294=1203.865,51.530,-46.205,-179.201,5.690,148.766
C04295=1203.870,51.281,-46.188,-179.203,5.689,148.767
C04296=1203.875,51.032,-46.172,-179.206,5.689,148.767
C04297=1203.879,50.782,-46.156,-179.209,5.687,148.768
C04298=1203.885,50.533,-46.139,-179.212,5.687,148.769
C04299=1203.890,50.282,-46.123,-179.214,5.686,148.769
C04300=1203.895,50.034,-46.106,-179.216,5.685,148.770
C04301=1203.900,49.784,-46.091,-179.219,5.685,148.770
C04302=1203.905,49.535,-46.074,-179.222,5.684,148.771
C04303=1203.910,49.285,-46.058,-179.224,5.683,148.772
C04304=1203.915,49.036,-46.042,-179.226,5.683,148.772
C04305=1203.920,48.786,-46.026,-179.229,5.682,148.773
C04306=1203.925,48.537,-46.010,-179.232,5.682,148.774
C04307=1203.930,48.288,-45.994,-179.234,5.681,148.774
C04308=1203.935,48.038,-45.977,-179.236,5.680,148.775
C04309=1203.940,47.789,-45.962,-179.240,5.679,148.775
C04310=1203.944,47.539,-45.945,-179.242,5.678,148.776
C04311=1203.950,47.290,-45.930,-179.244,5.677,148.776
C04312=1203.954,47.040,-45.913,-179.247,5.677,148.777
C04313=1203.960,46.791,-45.897,-179.250,5.676,148.778
C04314=1203.964,46.542,-45.881,-179.252,5.676,148.778
C04315=1203.969,46.292,-45.865,-179.255,5.675,148.779
C04316=1203.974,46.043,-45.848,-179.257,5.674,148.780
C04317=1203.979,45.793,-45.833,-179.260,5.674,148.780
C04318=1203.985,45.544,-45.817,-179.262,5.673,148.781
C04319=1203.988,45.295,-45.801,-179.265,5.672,148.781
C04320=1203.994,45.045,-45.786,-179.267,5.672,148.782
C04321=1203.999,44.795,-45.770,-179.270,5.671,148.783
C04322=1204.004,44.546,-45.753,-179.273,5.671,148.783
C04323=1204.009,44.297,-45.738,-179.275,5.669,148.784
C04324=1204.014,44.047,-45.721,-179.278,5.669,148.784
C04325=1204.019,43.798,-45.706,-179.281,5.668,148.785
C04326=1204.024,43.548,-45.690,-179.283,5.668,148.786
C04327=1204.029,43.299,-45.673,-179.285,5.667,148.786
C04328=1204.034,43.050,-45.658,-179.288,5.666,148.787
C04329=1204.039,42.800,-45.642,-179.291,5.666,148.788
C04330=1204.044,42.551,-45.627,-179.293,5.665,148.788
C04331=1204.048,42.301,-45.610,-179.295,5.664,148.789
C04332=1204.054,42.052,-45.594,-179.298,5.664,148.789
C04333=1204.059,41.802,-45.579,-179.301,5.663,148.790
C04334=1204.063,41.553,-45.562,-179.303,5.663,148.791
C04335=1204.069,41.303,-45.547,-179.306,5.662,148.791
C04336=1204.073,41.054,-45.532,-179.308,5.661,148.792
C04337=1204.078,40.804,-45.516,-179.311,5.661,148.793
C04338=1204.084,40.555,-45.500,-179.313,5.660,148.793
C04339=1204.089,40.306,-45.484,-179.316,5.659,148.794
C04340=1204.093,40.056,-45.468,-179.318,5.659,148.794
C04341=1204.099,39.807,-45.452,-179.321,5.658,148.795
C04342=1204.104,39.557,-45.437,-179.323,5.658,148.796
C04343=1204.108,39.307,-45.421,-179.327,5.656,148.796
C04344=1204.113,39.059,-45.405,-179.329,5.655,148.797
C04345=1204.119,38.809,-45.389,-179.331,5.655,148.797
C04346=1204.124,38.559,-45.373,-179.334,5.654,148.798
C04347=1204.128,38.310,-45.358,-179.337,5.654,148.799
C04348=1204.134,38.061,-45.343,-179.339,5.653,148.799
C04349=1204.138,37.810,-45.327,-179.342,5.652,148.800
C04350=1204.143,37.562,-45.311,-179.344,5.652,148.801
C04351=1204.148,37.313,-45.296,-179.347,5.651,148.801
C04352=1204.153,37.062,-45.280,-179.349,5.651,148.802
C04353=1204.158,36.813,-45.264,-179.352,5.650,148.802
C04354=1204.164,36.564,-45.248,-179.354,5.649,148.803
C04355=1204.168,36.315,-45.233,-179.357,5.649,148.804
C04356=1204.173,36.064,-45.218,-179.360,5.648,148.804
C04357=1204.179,35.815,-45.202,-179.362,5.648,148.805
C04358=1204.183,35.566,-45.187,-179.364,5.647,148.806
C04359=1204.188,35.316,-45.171,-179.367,5.646,148.806
C04360=1204.193,35.066,-45.155,-179.370,5.646,148.807
C04361=1204.199,34.817,-45.140,-179.372,5.645,148.808
C04362=1204.203,34.568,-45.125,-179.374,5.644,148.808
C04363=1204.208,34.318,-45.109,-179.377,5.644,148.809
C04364=1204.214,34.068,-45.093,-179.380,5.643,148.809
C04365=1204.218,33.819,-45.078,-179.382,5.643,148.810
C04366=1204.224,33.570,-45.063,-179.385,5.642,148.811
C04367=1204.228,33.320,-45.047,-179.387,5.641,148.811
C04368=1204.233,33.071,-45.032,-179.390,5.641,148.812
C04369=1204.238,32.821,-45.016,-179.392,5.640,148.813
C04370=1204.243,32.572,-45.001,-179.395,5.640,148.813
C04371=1204.248,32.323,-44.986,-179.398,5.639,148.814
C04372=1204.253,32.073,-44.970,-179.400,5.638,148.814
C04373=1204.258,31.824,-44.955,-179.403,5.638,148.815
C04374=1204.263,31.574,-44.939,-179.405,5.637,148.816
C04375=1204.269,31.325,-44.923,-179.408,5.637,148.816
C04376=1204.273,31.075,-44.908,-179.410,5.636,148.817
C04377=1204.278,30.826,-44.893,-179.413,5.635,148.817
C04378=1204.283,30.577,-44.878,-179.415,5.635,148.818
C04379=1204.288,30.327,-44.862,-179.418,5.634,148.819
C04380=1204.293,30.077,-44.848,-179.421,5.634,148.820
C04381=1204.298,29.828,-44.832,-179.423,5.633,148.820
C04382=1204.303,29.578,-44.816,-179.425,5.632,148.821
C04383=1204.308,29.310,-44.800,-179.428,5.632,148.821
C04384=1204.314,29.041,-44.783,-179.431,5.631,148.822
C04385=1204.319,28.773,-44.767,-179.433,5.631,148.823
C04386=1204.325,28.503,-44.751,-179.437,5.629,148.823
C04387=1204.330,28.254,-44.735,-179.439,5.629,148.824
C04388=1204.335,28.005,-44.720,-179.441,5.629,148.825
C04389=1204.340,27.755,-44.705,-179.444,5.629,148.825
C04390=1204.345,27.506,-44.690,-179.447,5.628,148.826
C04391=1204.350,27.256,-44.674,-179.449,5.627,148.827
C04392=1204.354,27.007,-44.659,-179.451,5.627,148.827
C04393=1204.360,26.757,-44.644,-179.454,5.626,148.828
C04394=1204.365,26.508,-44.629,-179.457,5.626,148.829
C04395=1204.370,26.258,-44.614,-179.459,5.625,148.829
C04396=1204.375,26.009,-44.599,-179.461,5.624,148.830
C04397=1204.380,25.760,-44.583,-179.464,5.624,148.830
C04398=1204.385,25.509,-44.569,-179.467,5.623,148.831
C04399=1204.390,25.260,-44.553,-179.469,5.623,148.832
C04400=1204.395,25.011,-44.538,-179.472,5.622,148.832
C04401=1204.400,24.761,-44.524,-179.474,5.621,148.833
C04402=1204.405,24.512,-44.508,-179.477,5.621,148.834
C04403=1204.410,24.263,-44.493,-179.479,5.620,148.834
C04404=1204.415,24.012,-44.478,-179.482,5.620,148.835
C04405=1204.420,23.763,-44.463,-179.485,5.619,148.836
C04406=1204.425,23.514,-44.448,-179.487,5.619,148.836
C04407=1204.430,23.264,-44.433,-179.490,5.618,148.837
C04408=1204.434,23.014,-44.418,-179.492,5.617,148.837
C04409=1204.440,22.765,-44.402,-179.495,5.617,148.838
C04410=1204.445,22.515,-44.388,-179.497,5.616,148.839
C04411=1204.450,22.266,-44.373,-179.500,5.616,148.839
C04412=1204.455,22.016,-44.358,-179.502,5.615,148.840
C04413=1204.460,21.767,-44.343,-179.505,5.614,148.841
C04414=1204.465,21.518,-44.328,-179.508,5.614,148.841
C04415=1204.470,21.268,-44.313,-179.510,5.614,148.842
C04416=1204.475,21.019,-44.298,-179.512,5.614,148.843
C04417=1204.480,20.769,-44.284,-179.515,5.613,148.843
C04418=1204.485,20.520,-44.269,-179.517,5.612,148.844
C04419=1204.490,20.270,-44.254,-179.520,5.612,148.844
C04420=1204.495,20.021,-44.239,-179.522,5.611,148.845
C04421=1204.500,19.771,-44.224,-179.525,5.611,148.846
C04422=1204.506,19.522,-44.209,-179.528,5.610,148.846
C04423=1204.510,19.273,-44.194,-179.530,5.609,148.847
C04424=1204.515,19.023,-44.180,-179.532,5.609,148.848
C04425=1204.520,18.774,-44.165,-179.535,5.608,148.848
C04426=1204.526,18.524,-44.150,-179.538,5.608,148.849
C04427=1204.531,18.274,-44.135,-179.540,5.607,148.850
C04428=1204.535,18.025,-44.121,-179.543,5.607,148.850
C04429=1204.541,17.775,-44.106,-179.545,5.606,148.851
C04430=1204.546,17.526,-44.091,-179.548,5.605,148.851
C04431=1204.550,17.276,-44.076,-179.551,5.605,148.852
C04432=1204.555,17.027,-44.061,-179.553,5.605,148.853
C04433=1204.561,16.777,-44.046,-179.555,5.605,148.854
C04434=1204.565,16.528,-44.032,-179.558,5.604,148.854
C04435=1204.570,16.278,-44.017,-179.560,5.603,148.855
C04436=1204.575,16.028,-44.003,-179.563,5.603,148.855
C04437=1204.581,15.779,-43.987,-179.565,5.602,148.856
C04438=1204.586,15.529,-43.973,-179.568,5.602,148.857
C04439=1204.590,15.280,-43.958,-179.571,5.601,148.857
C04440=1204.595,15.031,-43.944,-179.573,5.601,148.858
C04441=1204.601,14.781,-43.929,-179.575,5.600,148.859
C04442=1204.606,14.531,-43.914,-179.578,5.599,148.859
C04443=1204.611,14.282,-43.900,-179.581,5.599,148.860
C04444=1204.616,14.032,-43.885,-179.583,5.599,148.861
C04445=1204.620,13.783,-43.870,-179.585,5.599,148.861
C04446=1204.626,13.533,-43.856,-179.588,5.598,148.862
C04447=1204.631,13.283,-43.841,-179.590,5.597,148.862
C04448=1204.636,13.034,-43.826,-179.593,5.597,148.863
C04449=1204.641,12.785,-43.812,-179.596,5.596,148.864
C04450=1204.646,12.535,-43.798,-179.598,5.596,148.864
C04451=1204.651,12.286,-43.783,-179.601,5.595,148.865
C04452=1204.656,12.036,-43.768,-179.604,5.595,148.866
C04453=1204.661,11.787,-43.754,-179.606,5.594,148.866
C04454=1204.666,11.537,-43.740,-179.608,5.593,148.867
C04455=1204.671,11.288,-43.725,-179.610,5.594,148.868
C04456=1204.676,11.038,-43.710,-179.613,5.593,148.868
C04457=1204.681,10.788,-43.696,-179.616,5.593,148.869
C04458=1204.686,10.539,-43.682,-179.618,5.592,148.870
C04459=1204.692,10.290,-43.667,-179.621,5.591,148.870
C04460=1204.697,10.040,-43.652,-179.623,5.591,148.871
C04461=1204.702,9.791,-43.638,-179.626,5.590,148.872
C04462=1204.707,9.541,-43.624,-179.628,5.590,148.872
C04463=1204.712,9.291,-43.609,-179.631,5.589,148.873
C04464=1204.716,9.042,-43.595,-179.634,5.589,148.874
C04465=1204.721,8.792,-43.580,-179.635,5.589,148.874
C04466=1204.726,8.543,-43.566,-179.638,5.588,148.875
C04467=1204.732,8.294,-43.552,-179.641,5.588,148.875
C04468=1204.737,8.044,-43.538,-179.643,5.587,148.876
C04469=1204.742,7.794,-43.523,-179.646,5.587,148.877
C04470=1204.747,7.544,-43.509,-179.649,5.586,148.877
C04471=1204.752,7.295,-43.494,-179.651,5.586,148.878
C04472=1204.757,7.045,-43.479,-179.653,5.585,148.879
C04473=1204.762,6.796,-43.465,-179.656,5.585,148.879
C04474=1204.767,6.547,-43.451,-179.658,5.585,148.880
C04475=1204.772,6.297,-43.437,-179.661,5.584,148.881
C04476=1204.777,6.047,-43.423,-179.663,5.584,148.881
C04477=1204.782,5.797,-43.408,-179.666,5.583,148.882
C04478=1204.787,5.548,-43.394,-179.668,5.582,148.882
C04479=1204.793,5.299,-43.380,-179.671,5.582,148.883
C04480=1204.798,5.049,-43.366,-179.674,5.581,148.884
C04481=1204.803,4.799,-43.352,-179.676,5.582,148.885
C04482=1204.808,4.550,-43.337,-179.678,5.581,148.885
C04483=1204.813,4.300,-43.323,-179.681,5.581,148.886
C04484=1204.818,4.051,-43.309,-179.684,5.580,148.887
C04485=1204.823,3.801,-43.295,-179.686,5.579,148.887
C04486=1204.827,3.552,-43.281,-179.688,5.579,148.888
C04487=1204.833,3.283,-43.265,-179.691,5.578,148.888
C04488=1204.839,3.013,-43.250,-179.694,5.578,148.889
C04489=1204.844,2.744,-43.234,-179.696,5.577,148.890
C04490=1204.850,2.476,-43.220,-179.700,5.577,148.891
C04491=1204.855,2.226,-43.205,-179.702,5.576,148.891
C04492=1204.860,1.976,-43.191,-179.704,5.576,148.892
C04493=1204.864,1.727,-43.177,-179.706,5.576,148.893
C04494=1204.869,1.478,-43.163,-179.709,5.575,148.893
C04495=1204.874,1.228,-43.149,-179.712,5.575,148.894
C04496=1204.879,0.979,-43.135,-179.714,5.574,148.895
C04497=1204.884,0.729,-43.121,-179.717,5.574,148.895
C04498=1204.890,0.479,-43.107,-179.719,5.573,148.896
C04499=1204.895,0.229,-43.093,-179.722,5.573,148.896
C04500=1204.900,-0.020,-43.079,-179.724,5.573,148.897
C04501=1204.905,-0.270,-43.065,-179.727,5.572,148.898
C04502=1204.911,-0.519,-43.051,-179.729,5.572,148.899
C04503=1204.915,-0.768,-43.037,-179.732,5.571,148.899
C04504=1204.920,-1.018,-43.023,-179.735,5.571,148.900
C04505=1204.925,-1.267,-43.009,-179.737,5.570,148.900
C04506=1204.931,-1.517,-42.995,-179.739,5.570,148.901
C04507=1204.936,-1.767,-42.981,-179.741,5.570,148.902
C04508=1204.941,-2.016,-42.967,-179.744,5.569,148.902
C04509=1204.945,-2.266,-42.953,-179.747,5.569,148.903
C04510=1204.950,-2.515,-42.939,-179.749,5.568,148.904
C04511=1204.956,-2.766,-42.925,-179.752,5.568,148.905
C04512=1204.961,-3.015,-42.912,-179.754,5.567,148.905
C04513=1204.966,-3.264,-42.897,-179.756,5.567,148.906
C04514=1204.971,-3.514,-42.883,-179.759,5.567,148.906
C04515=1204.976,-3.763,-42.870,-179.762,5.566,148.907
C04516=1204.981,-4.013,-42.856,-179.764,5.566,148.908
C04517=1204.986,-4.263,-42.842,-179.767,5.565,148.908
C04518=1204.992,-4.512,-42.828,-179.770,5.565,148.909
C04519=1204.996,-4.761,-42.814,-179.771,5.565,148.910
C04520=1205.001,-5.011,-42.801,-179.774,5.564,148.910
C04521=1205.007,-5.260,-42.787,-179.776,5.564,148.911
C04522=1205.012,-5.510,-42.772,-179.779,5.563,148.912
C04523=1205.017,-5.761,-42.759,-179.782,5.563,148.912
C04524=1205.022,-6.009,-42.746,-179.784,5.562,148.913
C04525=1205.027,-6.259,-42.731,-179.786,5.563,148.914
C04526=1205.032,-6.508,-42.717,-179.789,5.562,148.914
C04527=1205.037,-6.758,-42.704,-179.791,5.561,148.915
C04528=1205.042,-7.008,-42.690,-179.794,5.561,148.916
C04529=1205.047,-7.257,-42.676,-179.797,5.560,148.916
C04530=1205.053,-7.507,-42.663,-179.799,5.561,148.917
C04531=1205.057,-7.756,-42.649,-179.801,5.560,148.918
C04532=1205.063,-8.006,-42.636,-179.804,5.560,148.918
C04533=1205.068,-8.256,-42.622,-179.807,5.559,148.919
C04534=1205.072,-8.504,-42.608,-179.809,5.558,148.919
C04535=1205.078,-8.755,-42.595,-179.811,5.558,148.920
C04536=1205.083,-9.005,-42.580,-179.814,5.558,148.921
C04537=1205.087,-9.253,-42.567,-179.816,5.558,148.922
C04538=1205.093,-9.504,-42.554,-179.819,5.557,148.922
C04539=1205.098,-9.753,-42.540,-179.822,5.557,148.923
C04540=1205.103,-10.003,-42.527,-179.824,5.556,148.924
C04541=1205.108,-10.252,-42.512,-179.826,5.556,148.924
C04542=1205.114,-10.502,-42.499,-179.828,5.556,148.925
C04543=1205.118,-10.751,-42.485,-179.831,5.555,148.925
C04544=1205.124,-11.001,-42.472,-179.834,5.555,148.926
C04545=1205.129,-11.251,-42.458,-179.836,5.554,148.927
C04546=1205.133,-11.499,-42.445,-179.838,5.554,148.928
C04547=1205.139,-11.750,-42.431,-179.841,5.554,148.928
C04548=1205.143,-11.999,-42.417,-179.844,5.553,148.929
C04549=1205.149,-12.249,-42.404,-179.846,5.553,148.929
C04550=1205.154,-12.498,-42.390,-179.849,5.552,148.930
C04551=1205.159,-12.748,-42.377,-179.851,5.552,148.931
C04552=1205.164,-12.997,-42.363,-179.853,5.552,148.931
C04553=1205.169,-13.247,-42.351,-179.856,5.551,148.932
C04554=1205.174,-13.497,-42.337,-179.859,5.551,148.933
C04555=1205.180,-13.746,-42.323,-179.861,5.551,148.934
C04556=1205.184,-13.996,-42.310,-179.863,5.551,148.934
C04557=1205.190,-14.245,-42.296,-179.866,5.550,148.935
C04558=1205.194,-14.495,-42.283,-179.868,5.549,148.935
C04559=1205.200,-14.744,-42.269,-179.871,5.549,148.936
C04560=1205.204,-14.994,-42.256,-179.874,5.549,148.937
C04561=1205.210,-15.244,-42.243,-179.876,5.549,148.937
C04562=1205.214,-15.493,-42.229,-179.878,5.548,148.938
C04563=1205.220,-15.743,-42.216,-179.881,5.548,148.939
C04564=1205.225,-15.992,-42.203,-179.883,5.547,148.939
C04565=1205.230,-16.242,-42.189,-179.885,5.547,148.940
C04566=1205.235,-16.492,-42.176,-179.888,5.547,148.941
C04567=1205.240,-16.741,-42.162,-179.890,5.546,148.941
C04568=1205.245,-16.991,-42.150,-179.893,5.546,148.942
C04569=1205.251,-17.241,-42.136,-179.896,5.545,148.943
C04570=1205.255,-17.490,-42.123,-179.898,5.546,148.944
C04571=1205.261,-17.740,-42.109,-179.901,5.545,148.944
C04572=1205.265,-17.990,-42.096,-179.903,5.544,148.945
C04573=1205.271,-18.239,-42.083,-179.905,5.544,148.945
C04574=1205.276,-18.489,-42.070,-179.907,5.544,148.946
C04575=1205.281,-18.738,-42.056,-179.910,5.544,148.947
C04576=1205.286,-18.988,-42.043,-179.913,5.543,148.947
C04577=1205.291,-19.237,-42.030,-179.915,5.543,148.948
C04578=1205.297,-19.487,-42.017,-179.918,5.542,148.949
C04579=1205.302,-19.737,-42.003,-179.920,5.543,148.950
C04580=1205.307,-19.986,-41.990,-179.922,5.542,148.950
C04581=1205.312,-20.236,-41.976,-179.925,5.541,148.951
C04582=1205.317,-20.485,-41.964,-179.928,5.541,148.951
C04583=1205.322,-20.735,-41.951,-179.930,5.541,148.952
C04584=1205.327,-20.984,-41.937,-179.932,5.541,148.953
C04585=1205.332,-21.234,-41.924,-179.935,5.540,148.953
C04586=1205.338,-21.484,-41.911,-179.938,5.540,148.954
C04587=1205.343,-21.733,-41.898,-179.940,5.540,148.955
C04588=1205.347,-21.983,-41.885,-179.942,5.539,148.955
C04589=1205.353,-22.232,-41.871,-179.945,5.539,148.956
C04590=1205.358,-22.482,-41.859,-179.947,5.538,148.957
C04591=1205.364,-22.752,-41.844,-179.950,5.538,148.957
C04592=1205.369,-23.021,-41.831,-179.952,5.538,148.958
C04593=1205.374,-23.291,-41.816,-179.955,5.538,148.959
C04594=1205.380,-23.560,-41.802,-179.958,5.537,148.960
C04595=1205.385,-23.810,-41.789,-179.960,5.537,148.960
C04596=1205.390,-24.059,-41.776,-179.963,5.536,148.961
C04597=1205.396,-24.309,-41.763,-179.965,5.536,148.962
C04598=1205.400,-24.558,-41.749,-179.967,5.536,148.962
C04599=1205.405,-24.808,-41.737,-179.970,5.536,148.963
C04600=1205.410,-25.058,-41.723,-179.973,5.535,148.964
C04601=1205.416,-25.307,-41.711,-179.975,5.535,148.964
C04602=1205.421,-25.557,-41.698,-179.977,5.535,148.965
C04603=1205.425,-25.807,-41.685,-179.980,5.534,148.966
C04604=1205.431,-26.056,-41.672,-179.982,5.534,148.966
C04605=1205.436,-26.306,-41.659,-179.984,5.534,148.967
C04606=1205.441,-26.556,-41.646,-179.987,5.533,148.968
C04607=1205.447,-26.805,-41.633,-179.990,5.533,148.968
C04608=1205.452,-27.055,-41.621,-179.992,5.532,148.969
C04609=1205.456,-27.305,-41.608,-179.994,5.533,148.970
C04610=1205.461,-27.554,-41.595,-179.997,5.532,148.970
C04611=1205.467,-27.804,-41.582,-179.999,5.531,148.971
C04612=1205.471,-28.053,-41.568,179.998,5.531,148.972
C04613=1205.477,-28.302,-41.556,179.996,5.531,148.972
C04614=1205.482,-28.552,-41.543,179.993,5.531,148.973
C04615=1205.487,-28.802,-41.529,179.991,5.530,148.974
C04616=1205.492,-29.052,-41.517,179.988,5.530,148.974
C04617=1205.498,-29.301,-41.505,179.986,5.530,148.975
C04618=1205.502,-29.551,-41.492,179.983,5.530,148.976
C04619=1205.508,-29.801,-41.479,179.981,5.529,148.976
C04620=1205.513,-30.050,-41.466,179.978,5.528,148.977
C04621=1205.518,-30.300,-41.454,179.976,5.529,148.978
C04622=1205.523,-30.550,-41.441,179.974,5.528,148.978
C04623=1205.528,-30.799,-41.428,179.971,5.528,148.979
C04624=1205.534,-31.049,-41.415,179.969,5.528,148.980
C04625=1205.538,-31.299,-41.402,179.966,5.528,148.980
C04626=1205.543,-31.548,-41.389,179.964,5.527,148.981
C04627=1205.548,-31.797,-41.377,179.961,5.527,148.982
C04628=1205.554,-32.046,-41.364,179.959,5.527,148.982
C04629=1205.559,-32.297,-41.350,179.957,5.526,148.983
C04630=1205.564,-32.547,-41.339,179.954,5.526,148.984
C04631=1205.569,-32.796,-41.326,179.952,5.526,148.984
C04632=1205.575,-33.045,-41.313,179.949,5.526,148.985
C04633=1205.579,-33.295,-41.300,179.947,5.525,148.986
C04634=1205.584,-33.545,-41.288,179.944,5.525,148.986
C04635=1205.589,-33.794,-41.275,179.942,5.525,148.987
C04636=1205.595,-34.044,-41.262,179.940,5.524,148.988
C04637=1205.600,-34.294,-41.250,179.937,5.524,148.988
C04638=1205.605,-34.544,-41.237,179.935,5.524,148.989
C04639=1205.610,-34.793,-41.225,179.932,5.524,148.990
C04640=1205.615,-35.042,-41.212,179.930,5.523,148.990
C04641=1205.620,-35.292,-41.199,179.927,5.523,148.991
C04642=1205.625,-35.542,-41.187,179.925,5.523,148.992
C04643=1205.630,-35.792,-41.174,179.922,5.523,148.993
C04644=1205.636,-36.041,-41.162,179.920,5.522,148.993
C04645=1205.641,-36.290,-41.149,179.918,5.522,148.994
C04646=1205.647,-36.540,-41.137,179.915,5.522,148.994
C04647=1205.651,-36.790,-41.124,179.913,5.521,148.995
C04648=1205.656,-37.040,-41.111,179.910,5.521,148.996
C04649=1205.662,-37.289,-41.099,179.908,5.521,148.997
C04650=1205.667,-37.539,-41.087,179.905,5.521,148.997
C04651=1205.672,-37.788,-41.074,179.903,5.520,148.998
C04652=1205.677,-38.038,-41.061,179.901,5.520,148.998
C04653=1205.682,-38.288,-41.049,179.898,5.520,148.999
C04654=1205.687,-38.538,-41.037,179.896,5.519,149.000
C04655=1205.692,-38.787,-41.024,179.894,5.519,149.000
C04656=1205.697,-39.036,-41.011,179.891,5.519,149.001
C04657=1205.703,-39.286,-41.000,179.888,5.518,149.002
C04658=1205.708,-39.535,-40.987,179.886,5.519,149.003
C04659=1205.713,-39.785,-40.974,179.884,5.518,149.003
C04660=1205.718,-40.035,-40.962,179.881,5.518,149.004
C04661=1205.723,-40.285,-40.950,179.879,5.517,149.004
C04662=1205.728,-40.534,-40.937,179.877,5.517,149.005
C04663=1205.734,-40.784,-40.925,179.874,5.517,149.006
C04664=1205.739,-41.033,-40.912,179.871,5.516,149.007
C04665=1205.744,-41.284,-40.900,179.869,5.517,149.007
C04666=1205.749,-41.533,-40.888,179.867,5.516,149.008
C04667=1205.754,-41.783,-40.875,179.864,5.516,149.009
C04668=1205.759,-42.033,-40.863,179.862,5.516,149.009
C04669=1205.764,-42.282,-40.851,179.860,5.515,149.010
C04670=1205.770,-42.532,-40.839,179.857,5.515,149.011
C04671=1205.775,-42.781,-40.826,179.855,5.515,149.011
C04672=1205.780,-43.030,-40.813,179.852,5.515,149.012
C04673=1205.786,-43.280,-40.802,179.850,5.514,149.013
C04674=1205.790,-43.530,-40.789,179.848,5.515,149.013
C04675=1205.795,-43.780,-40.777,179.845,5.514,149.014
C04676=1205.801,-44.030,-40.764,179.843,5.513,149.015
C04677=1205.806,-44.280,-40.752,179.841,5.514,149.015
C04678=1205.810,-44.529,-40.740,179.838,5.513,149.016
C04679=1205.816,-44.779,-40.728,179.835,5.513,149.017
C04680=1205.821,-45.028,-40.716,179.833,5.512,149.017
C04681=1205.826,-45.278,-40.704,179.831,5.513,149.018
C04682=1205.832,-45.527,-40.691,179.828,5.512,149.019
C04683=1205.837,-45.777,-40.679,179.826,5.511,149.019
C04684=1205.842,-46.026,-40.667,179.824,5.512,149.020
C04685=1205.848,-46.276,-40.655,179.821,5.511,149.021
C04686=1205.853,-46.526,-40.642,179.818,5.511,149.021
C04687=1205.857,-46.776,-40.631,179.816,5.511,149.022
C04688=1205.862,-47.025,-40.618,179.814,5.511,149.023
C04689=1205.867,-47.275,-40.606,179.811,5.510,149.023
C04690=1205.873,-47.525,-40.594,179.809,5.511,149.024
C04691=1205.878,-47.774,-40.582,179.807,5.510,149.025
C04692=1205.883,-48.024,-40.570,179.804,5.509,149.025
C04693=1205.888,-48.273,-40.558,179.802,5.510,149.026
C04694=1205.893,-48.523,-40.546,179.799,5.509,149.027
C04695=1205.899,-48.793,-40.533,179.797,5.509,149.027
C04696=1205.905,-49.064,-40.520,179.794,5.509,149.028
C04697=1205.910,-49.333,-40.506,179.792,5.509,149.029
C04698=1205.916,-49.603,-40.493,179.789,5.508,149.030
C04699=1205.921,-49.853,-40.482,179.786,5.508,149.030
C04700=1205.926,-50.103,-40.470,179.784,5.508,149.031
C04701=1205.931,-50.352,-40.458,179.782,5.508,149.032
C04702=1205.937,-50.602,-40.446,179.779,5.507,149.032
C04703=1205.942,-50.851,-40.433,179.777,5.507,149.033
C04704=1205.947,-51.101,-40.421,179.774,5.507,149.034
C04705=1205.952,-51.351,-40.410,179.772,5.506,149.034
C04706=1205.957,-51.601,-40.398,179.770,5.507,149.035
C04707=1205.962,-51.850,-40.385,179.767,5.506,149.036
C04708=1205.968,-52.100,-40.374,179.765,5.506,149.036
C04709=1205.973,-52.350,-40.362,179.763,5.506,149.037
C04710=1205.978,-52.599,-40.350,179.760,5.506,149.038
C04711=1205.983,-52.849,-40.338,179.757,5.505,149.038
C04712=1205.988,-53.098,-40.327,179.755,5.505,149.039
C04713=1205.993,-53.348,-40.315,179.753,5.505,149.040
C04714=1205.998,-53.598,-40.302,179.751,5.505,149.040
C04715=1206.004,-53.848,-40.290,179.748,5.504,149.041
C04716=1206.008,-54.097,-40.279,179.746,5.504,149.042
C04717=1206.014,-54.347,-40.267,179.743,5.504,149.042
C04718=1206.019,-54.596,-40.254,179.741,5.504,149.043
C04719=1206.024,-54.846,-40.243,179.738,5.503,149.044
C04720=1206.029,-55.096,-40.231,179.737,5.503,149.044
C04721=1206.035,-55.346,-40.219,179.734,5.503,149.045
C04722=1206.039,-55.595,-40.207,179.731,5.503,149.046
C04723=1206.044,-55.845,-40.195,179.729,5.503,149.046
C04724=1206.050,-56.095,-40.184,179.726,5.502,149.047
C04725=1206.054,-56.344,-40.172,179.724,5.503,149.048
C04726=1206.061,-56.594,-40.161,179.722,5.502,149.049
C04727=1206.066,-56.844,-40.149,179.720,5.502,149.049
C04728=1206.070,-57.093,-40.137,179.717,5.502,149.050
C04729=1206.076,-57.343,-40.125,179.715,5.501,149.050
C04730=1206.081,-57.593,-40.113,179.712,5.501,149.051
C04731=1206.086,-57.842,-40.102,179.710,5.501,149.052
C04732=1206.091,-58.092,-40.090,179.707,5.501,149.053
C04733=1206.096,-58.342,-40.079,179.705,5.500,149.053
C04734=1206.101,-58.592,-40.067,179.703,5.500,149.054
C04735=1206.107,-58.842,-40.055,179.700,5.500,149.054
C04736=1206.111,-59.091,-40.043,179.698,5.500,149.055
C04737=1206.117,-59.340,-40.031,179.696,5.500,149.056
C04738=1206.122,-59.589,-40.020,179.693,5.499,149.057
C04739=1206.127,-59.839,-40.008,179.691,5.500,149.057
C04740=1206.133,-60.089,-39.996,179.688,5.499,149.058
C04741=1206.138,-60.339,-39.985,179.686,5.498,149.058
C04742=1206.143,-60.589,-39.973,179.684,5.499,149.059
C04743=1206.148,-60.839,-39.962,179.681,5.498,149.060
C04744=1206.153,-61.088,-39.950,179.679,5.499,149.061
C04745=1206.158,-61.337,-39.939,179.677,5.498,149.061
C04746=1206.164,-61.587,-39.927,179.674,5.498,149.062
C04747=1206.168,-61.837,-39.916,179.672,5.498,149.063
C04748=1206.174,-62.087,-39.904,179.670,5.497,149.063
C04749=1206.179,-62.337,-39.892,179.668,5.498,149.064
C04750=1206.184,-62.586,-39.881,179.665,5.497,149.065
C04751=1206.190,-62.836,-39.869,179.662,5.497,149.065
C04752=1206.195,-63.085,-39.858,179.660,5.497,149.066
C04753=1206.200,-63.335,-39.846,179.657,5.497,149.067
C04754=1206.205,-63.585,-39.835,179.655,5.496,149.067
C04755=1206.210,-63.835,-39.823,179.653,5.496,149.068
C04756=1206.215,-64.084,-39.812,179.651,5.496,149.069
C04757=1206.221,-64.334,-39.800,179.648,5.496,149.069
C04758=1206.226,-64.583,-39.789,179.646,5.496,149.070
C04759=1206.231,-64.833,-39.777,179.643,5.495,149.071
C04760=1206.236,-65.083,-39.766,179.641,5.496,149.071
C04761=1206.241,-65.333,-39.754,179.639,5.495,149.072
C04762=1206.247,-65.582,-39.744,179.637,5.495,149.073
C04763=1206.252,-65.832,-39.732,179.634,5.495,149.073
C04764=1206.257,-66.082,-39.720,179.631,5.494,149.074
C04765=1206.262,-66.332,-39.709,179.629,5.495,149.075
C04766=1206.267,-66.581,-39.697,179.627,5.494,149.075
C04767=1206.272,-66.830,-39.686,179.625,5.495,149.076
C04768=1206.278,-67.080,-39.674,179.622,5.494,149.077
C04769=1206.283,-67.330,-39.663,179.620,5.493,149.077
C04770=1206.288,-67.580,-39.651,179.618,5.494,149.078
C04771=1206.294,-67.829,-39.641,179.615,5.493,149.079
C04772=1206.298,-68.079,-39.630,179.613,5.494,149.079
C04773=1206.304,-68.329,-39.618,179.610,5.493,149.080
C04774=1206.308,-68.579,-39.606,179.608,5.492,149.081
C04775=1206.314,-68.828,-39.595,179.606,5.493,149.081
C04776=1206.319,-69.078,-39.584,179.603,5.492,149.082
C04777=1206.325,-69.328,-39.573,179.601,5.493,149.083
C04778=1206.330,-69.578,-39.561,179.599,5.492,149.083
C04779=1206.335,-69.827,-39.550,179.596,5.492,149.084
C04780=1206.340,-70.077,-39.538,179.594,5.492,149.085
C04781=1206.345,-70.327,-39.528,179.592,5.491,149.085
C04782=1206.351,-70.576,-39.517,179.590,5.492,149.086
C04783=1206.356,-70.826,-39.505,179.587,5.491,149.087
C04784=1206.361,-71.075,-39.494,179.584,5.491,149.087
C04785=1206.366,-71.326,-39.483,179.582,5.491,149.088
C04786=1206.372,-71.575,-39.472,179.579,5.491,149.089
C04787=1206.376,-71.824,-39.460,179.578,5.491,149.089
C04788=1206.382,-72.074,-39.448,179.575,5.490,149.090
C04789=1206.387,-72.324,-39.438,179.573,5.490,149.091
C04790=1206.392,-72.573,-39.427,179.570,5.490,149.091
C04791=1206.398,-72.823,-39.415,179.568,5.490,149.092
C04792=1206.403,-73.074,-39.405,179.566,5.490,149.093
C04793=1206.408,-73.323,-39.394,179.563,5.489,149.093
C04794=1206.413,-73.572,-39.382,179.561,5.490,149.094
C04795=1206.418,-73.823,-39.371,179.559,5.489,149.095
C04796=1206.424,-74.072,-39.360,179.556,5.489,149.095
C04797=1206.428,-74.321,-39.349,179.554,5.489,149.096
C04798=1206.434,-74.572,-39.338,179.551,5.489,149.097
C04799=1206.440,-74.842,-39.326,179.549,5.489,149.098
C04800=1206.445,-75.113,-39.314,179.547,5.489,149.098
C04801=1206.451,-75.382,-39.302,179.544,5.488,149.099
C04802=1206.457,-75.653,-39.289,179.541,5.488,149.100
C04803=1206.462,-75.904,-39.279,179.539,5.488,149.100
C04804=1206.467,-76.153,-39.268,179.537,5.487,149.101
C04805=1206.473,-76.403,-39.257,179.535,5.488,149.102
C04806=1206.477,-76.653,-39.245,179.532,5.487,149.102
C04807=1206.483,-76.902,-39.234,179.530,5.488,149.103
C04808=1206.488,-77.152,-39.224,179.527,5.487,149.104
C04809=1206.493,-77.402,-39.212,179.525,5.487,149.104
C04810=1206.499,-77.651,-39.202,179.523,5.487,149.105
C04811=1206.503,-77.901,-39.191,179.520,5.486,149.106
C04812=1206.509,-78.151,-39.180,179.518,5.487,149.106
C04813=1206.514,-78.401,-39.168,179.516,5.486,149.107
C04814=1206.519,-78.651,-39.158,179.514,5.487,149.108
C04815=1206.525,-78.900,-39.147,179.511,5.486,149.108
C04816=1206.530,-79.150,-39.136,179.509,5.485,149.109
C04817=1206.535,-79.399,-39.125,179.507,5.486,149.110
C04818=1206.540,-79.649,-39.114,179.504,5.485,149.110
C04819=1206.545,-79.899,-39.103,179.502,5.486,149.111
C04820=1206.551,-80.148,-39.092,179.499,5.485,149.112
C04821=1206.556,-80.398,-39.081,179.498,5.485,149.112
C04822=1206.561,-80.647,-39.071,179.495,5.485,149.113
C04823=1206.566,-80.897,-39.060,179.492,5.484,149.114
C04824=1206.572,-81.148,-39.049,179.490,5.485,149.114
C04825=1206.577,-81.397,-39.038,179.488,5.484,149.115
C04826=1206.582,-81.647,-39.027,179.486,5.484,149.116
C04827=1206.587,-81.896,-39.016,179.483,5.484,149.116
C04828=1206.592,-82.146,-39.006,179.481,5.484,149.117
C04829=1206.597,-82.396,-38.995,179.479,5.484,149.118
C04830=1206.603,-82.645,-38.984,179.476,5.484,149.118
C04831=1206.607,-82.895,-38.973,179.474,5.484,149.119
C04832=1206.614,-83.145,-38.962,179.472,5.483,149.120
C04833=1206.619,-83.395,-38.952,179.470,5.483,149.120
C04834=1206.624,-83.644,-38.941,179.467,5.483,149.121
C04835=1206.629,-83.894,-38.930,179.465,5.483,149.122
C04836=1206.634,-84.143,-38.919,179.462,5.483,149.122
C04837=1206.639,-84.394,-38.909,179.460,5.483,149.123
C04838=1206.644,-84.644,-38.898,179.458,5.482,149.124
C04839=1206.649,-84.893,-38.887,179.456,5.483,149.124
C04840=1206.654,-85.143,-38.877,179.453,5.482,149.125
C04841=1206.660,-85.392,-38.866,179.450,5.482,149.126
C04842=1206.665,-85.642,-38.855,179.449,5.482,149.126
C04843=1206.670,-85.892,-38.845,179.446,5.481,149.127
C04844=1206.675,-86.142,-38.834,179.444,5.482,149.128
C04845=1206.681,-86.391,-38.823,179.441,5.481,149.128
C04846=1206.686,-86.641,-38.812,179.439,5.482,149.129
C04847=1206.692,-86.891,-38.802,179.437,5.481,149.130
C04848=1206.697,-87.141,-38.791,179.435,5.481,149.130
C04849=1206.702,-87.390,-38.780,179.432,5.481,149.131
C04850=1206.707,-87.640,-38.770,179.430,5.481,149.132
C04851=1206.713,-87.889,-38.759,179.428,5.481,149.132
C04852=1206.718,-88.139,-38.748,179.425,5.480,149.133
C04853=1206.723,-88.389,-38.738,179.423,5.480,149.134
C04854=1206.728,-88.639,-38.728,179.421,5.480,149.134
C04855=1206.733,-88.888,-38.717,179.419,5.480,149.135
C04856=1206.738,-89.138,-38.706,179.416,5.480,149.136
C04857=1206.744,-89.388,-38.696,179.414,5.480,149.136
C04858=1206.749,-89.638,-38.685,179.412,5.479,149.137
C04859=1206.754,-89.887,-38.674,179.409,5.480,149.138
C04860=1206.759,-90.137,-38.664,179.407,5.479,149.138
C04861=1206.765,-90.387,-38.654,179.405,5.480,149.139
C04862=1206.770,-90.636,-38.643,179.403,5.479,149.140
C04863=1206.775,-90.887,-38.633,179.400,5.479,149.140
C04864=1206.780,-91.135,-38.623,179.398,5.479,149.141
C04865=1206.785,-91.386,-38.612,179.395,5.478,149.142
C04866=1206.791,-91.635,-38.602,179.393,5.479,149.142
C04867=1206.796,-91.885,-38.591,179.391,5.478,149.143
C04868=1206.801,-92.135,-38.581,179.389,5.478,149.144
C04869=1206.806,-92.385,-38.570,179.386,5.478,149.144
C04870=1206.812,-92.634,-38.559,179.384,5.478,149.145
C04871=1206.817,-92.884,-38.549,179.382,5.478,149.145
C04872=1206.822,-93.134,-38.539,179.380,5.478,149.146
C04873=1206.828,-93.383,-38.528,179.377,5.477,149.147
C04874=1206.833,-93.634,-38.518,179.375,5.478,149.148
C04875=1206.838,-93.883,-38.508,179.372,5.477,149.148
C04876=1206.844,-94.133,-38.497,179.371,5.477,149.149
C04877=1206.849,-94.382,-38.486,179.368,5.477,149.150
C04878=1206.853,-94.632,-38.477,179.366,5.477,149.150
C04879=1206.858,-94.882,-38.466,179.363,5.477,149.151
C04880=1206.864,-95.131,-38.456,179.362,5.477,149.151
C04881=1206.870,-95.381,-38.446,179.359,5.477,149.152
C04882=1206.875,-95.631,-38.435,179.357,5.477,149.153
C04883=1206.880,-95.881,-38.425,179.354,5.477,149.154
C04884=1206.885,-96.131,-38.414,179.352,5.476,149.154
C04885=1206.891,-96.381,-38.404,179.350,5.476,149.155
C04886=1206.896,-96.630,-38.394,179.347,5.476,149.155
C04887=1206.901,-96.880,-38.384,179.345,5.476,149.156
C04888=1206.906,-97.130,-38.374,179.342,5.476,149.157
C04889=1206.912,-97.379,-38.363,179.341,5.476,149.157
C04890=1206.917,-97.629,-38.353,179.338,5.475,149.158
C04891=1206.923,-97.879,-38.343,179.336,5.476,149.159
C04892=1206.927,-98.129,-38.333,179.333,5.475,149.160
C04893=1206.932,-98.378,-38.322,179.332,5.475,149.160
C04894=1206.938,-98.628,-38.312,179.329,5.475,149.161
C04895=1206.943,-98.878,-38.302,179.327,5.475,149.161
C04896=1206.949,-99.128,-38.291,179.324,5.475,149.162
C04897=1206.953,-99.377,-38.282,179.322,5.475,149.163
C04898=1206.958,-99.627,-38.271,179.320,5.474,149.163
C04899=1206.964,-99.877,-38.261,179.318,5.475,149.164
C04900=1206.970,-100.126,-38.251,179.315,5.474,149.165
C04901=1206.975,-100.376,-38.240,179.313,5.475,149.165
C04902=1206.979,-100.626,-38.231,179.311,5.474,149.166
C04903=1206.985,-100.897,-38.219,179.309,5.474,149.167
C04904=1206.991,-101.168,-38.209,179.306,5.474,149.167
C04905=1206.997,-101.440,-38.197,179.304,5.473,149.168
C04906=1207.003,-101.711,-38.187,179.302,5.474,149.169
C04907=1207.008,-101.961,-38.177,179.299,5.473,149.170
C04908=1207.013,-102.210,-38.167,179.297,5.474,149.170
C04909=1207.018,-102.460,-38.156,179.294,5.473,149.171
C04910=1207.024,-102.710,-38.146,179.293,5.473,149.171
C04911=1207.029,-102.960,-38.136,179.290,5.473,149.172
C04912=1207.034,-103.209,-38.126,179.288,5.473,149.173
C04913=1207.039,-103.459,-38.116,179.285,5.473,149.174
C04914=1207.045,-103.709,-38.106,179.283,5.473,149.174
C04915=1207.049,-103.959,-38.096,179.281,5.472,149.175
C04916=1207.055,-104.209,-38.086,179.279,5.473,149.175
C04917=1207.060,-104.458,-38.076,179.276,5.472,149.176
C04918=1207.065,-104.707,-38.066,179.274,5.472,149.177
C04919=1207.070,-104.958,-38.056,179.272,5.472,149.177
C04920=1207.076,-105.207,-38.045,179.270,5.472,149.178
C04921=1207.082,-105.457,-38.036,179.267,5.472,149.179
C04922=1207.087,-105.707,-38.026,179.265,5.472,149.179
C04923=1207.092,-105.957,-38.016,179.263,5.472,149.180
C04924=1207.097,-106.206,-38.006,179.261,5.472,149.181
C04925=1207.102,-106.456,-37.997,179.258,5.472,149.181
C04926=1207.108,-106.706,-37.986,179.256,5.472,149.182
C04927=1207.112,-106.956,-37.977,179.254,5.471,149.183
C04928=1207.118,-107.205,-37.966,179.252,5.471,149.183
C04929=1207.124,-107.455,-37.956,179.249,5.471,149.184
C04930=1207.129,-107.705,-37.947,179.247,5.471,149.185
C04931=1207.134,-107.955,-37.937,179.245,5.471,149.185
C04932=1207.139,-108.204,-37.926,179.243,5.471,149.186
C04933=1207.144,-108.454,-37.918,179.240,5.470,149.186
C04934=1207.150,-108.704,-37.907,179.238,5.471,149.187
C04935=1207.155,-108.953,-37.898,179.236,5.470,149.188
C04936=1207.160,-109.203,-37.887,179.234,5.471,149.189
C04937=1207.166,-109.454,-37.878,179.231,5.470,149.189
C04938=1207.171,-109.703,-37.868,179.229,5.470,149.190
C04939=1207.176,-109.952,-37.858,179.227,5.470,149.191
C04940=1207.181,-110.202,-37.849,179.225,5.470,149.191
C04941=1207.186,-110.452,-37.838,179.222,5.469,149.192
C04942=1207.192,-110.702,-37.828,179.220,5.470,149.192
C04943=1207.197,-110.952,-37.819,179.218,5.469,149.193
C04944=1207.203,-111.201,-37.809,179.216,5.469,149.194
C04945=1207.208,-111.451,-37.799,179.213,5.469,149.194
C04946=1207.213,-111.701,-37.790,179.211,5.469,149.195
C04947=1207.218,-111.951,-37.780,179.208,5.469,149.196
C04948=1207.223,-112.200,-37.770,179.207,5.469,149.196
C04949=1207.229,-112.450,-37.760,179.204,5.469,149.197
C04950=1207.234,-112.700,-37.751,179.202,5.469,149.198
C04951=1207.240,-112.950,-37.741,179.200,5.468,149.198
C04952=1207.244,-113.200,-37.731,179.198,5.469,149.199
C04953=1207.250,-113.449,-37.721,179.195,5.468,149.200
C04954=1207.255,-113.699,-37.712,179.193,5.469,149.200
C04955=1207.261,-113.949,-37.702,179.191,5.468,149.201
C04956=1207.266,-114.198,-37.693,179.189,5.468,149.202
C04957=1207.271,-114.448,-37.683,179.186,5.468,149.202
C04958=1207.277,-114.698,-37.674,179.185,5.468,149.203
C04959=1207.282,-114.948,-37.663,179.182,5.467,149.203
C04960=1207.286,-115.197,-37.654,179.180,5.468,149.204
C04961=1207.292,-115.447,-37.644,179.178,5.467,149.205
C04962=1207.297,-115.697,-37.635,179.175,5.467,149.205
C04963=1207.303,-115.947,-37.625,179.173,5.468,149.206
C04964=1207.308,-116.196,-37.615,179.171,5.467,149.207
C04965=1207.314,-116.446,-37.606,179.169,5.467,149.207
C04966=1207.319,-116.696,-37.596,179.166,5.467,149.208
C04967=1207.324,-116.946,-37.586,179.164,5.467,149.209
C04968=1207.329,-117.196,-37.577,179.162,5.466,149.209
C04969=1207.334,-117.445,-37.568,179.160,5.467,149.210
C04970=1207.340,-117.695,-37.558,179.157,5.466,149.211
C04971=1207.345,-117.945,-37.549,179.156,5.466,149.211
C04972=1207.350,-118.194,-37.539,179.153,5.466,149.212
C04973=1207.356,-118.444,-37.530,179.151,5.466,149.213
C04974=1207.361,-118.694,-37.520,179.148,5.466,149.213
C04975=1207.366,-118.944,-37.511,179.147,5.466,149.214
C04976=1207.372,-119.193,-37.502,179.144,5.466,149.214
C04977=1207.377,-119.444,-37.491,179.142,5.466,149.215
C04978=1207.382,-119.694,-37.482,179.140,5.465,149.216
C04979=1207.387,-119.943,-37.472,179.138,5.466,149.216
C04980=1207.393,-120.193,-37.463,179.135,5.465,149.217
C04981=1207.397,-120.442,-37.454,179.133,5.465,149.218
C04982=1207.403,-120.692,-37.444,179.131,5.466,149.218
C04983=1207.408,-120.942,-37.435,179.129,5.465,149.219
C04984=1207.414,-121.192,-37.425,179.127,5.465,149.219
C04985=1207.419,-121.442,-37.416,179.124,5.465,149.220
C04986=1207.424,-121.691,-37.406,179.122,5.465,149.221
C04987=1207.430,-121.941,-37.397,179.120,5.464,149.221
C04988=1207.435,-122.191,-37.388,179.118,5.465,149.222
C04989=1207.440,-122.440,-37.378,179.115,5.464,149.223
C04990=1207.446,-122.690,-37.369,179.114,5.464,149.223
C04991=1207.451,-122.940,-37.360,179.111,5.464,149.224
C04992=1207.456,-123.189,-37.350,179.109,5.464,149.225
C04993=1207.462,-123.440,-37.341,179.107,5.464,149.225
C04994=1207.467,-123.689,-37.332,179.105,5.464,149.226
C04995=1207.472,-123.939,-37.322,179.103,5.464,149.227
C04996=1207.478,-124.189,-37.313,179.100,5.464,149.227
C04997=1207.483,-124.439,-37.304,179.098,5.464,149.228
C04998=1207.488,-124.688,-37.294,179.096,5.464,149.229
C04999=1207.493,-124.939,-37.285,179.094,5.464,149.229
C05000=1207.498,-125.189,-37.276,179.091,5.463,149.230
C05001=1207.503,-125.438,-37.267,179.089,5.464,149.231
C05002=1207.508,-125.688,-37.257,179.087,5.463,149.231
C05003=1207.514,-125.938,-37.248,179.085,5.463,149.232
C05004=1207.519,-126.188,-37.239,179.082,5.463,149.232
C05005=1207.525,-126.436,-37.229,179.081,5.463,149.233
C05006=1207.531,-126.686,-37.220,179.078,5.462,149.234
C05007=1207.109,-126.697,-37.258,179.074,5.466,149.236
C05008=1207.104,-126.448,-37.267,179.076,5.466,149.235
C05009=1207.098,-126.198,-37.277,179.078,5.466,149.234
C05010=1207.093,-125.948,-37.286,179.081,5.466,149.234
C05011=1207.087,-125.698,-37.295,179.083,5.466,149.233
C05012=1207.083,-125.449,-37.304,179.085,5.467,149.232
C05013=1207.077,-125.199,-37.314,179.087,5.467,149.232
C05014=1207.071,-124.949,-37.323,179.090,5.467,149.231
C05015=1207.066,-124.699,-37.331,179.092,5.467,149.230
C05016=1207.061,-124.450,-37.342,179.094,5.468,149.230
C05017=1207.056,-124.200,-37.351,179.096,5.467,149.229
C05018=1207.050,-123.950,-37.359,179.099,5.468,149.229
C05019=1207.045,-123.700,-37.370,179.100,5.468,149.228
C05020=1207.040,-123.451,-37.379,179.102,5.467,149.227
C05021=1207.034,-123.201,-37.387,179.105,5.468,149.227
C05022=1207.029,-122.951,-37.398,179.107,5.468,149.226
C05023=1207.024,-122.701,-37.407,179.109,5.468,149.225
C05024=1207.019,-122.451,-37.415,179.111,5.468,149.225
C05025=1207.013,-122.202,-37.426,179.114,5.468,149.224
C05026=1207.008,-121.952,-37.435,179.116,5.468,149.224
C05027=1207.003,-121.702,-37.443,179.118,5.468,149.223
C05028=1206.997,-121.453,-37.454,179.120,5.468,149.222
C05029=1206.992,-121.202,-37.463,179.123,5.469,149.222
C05030=1206.988,-120.953,-37.473,179.125,5.468,149.221
C05031=1206.982,-120.703,-37.482,179.127,5.469,149.220
C05032=1206.977,-120.453,-37.491,179.129,5.469,149.220
C05033=1206.972,-120.204,-37.501,179.132,5.469,149.219
C05034=1206.966,-119.953,-37.510,179.134,5.469,149.218
C05035=1206.961,-119.704,-37.520,179.135,5.469,149.218
C05036=1206.955,-119.454,-37.529,179.138,5.469,149.217
C05037=1206.950,-119.204,-37.538,179.140,5.469,149.216
C05038=1206.945,-118.955,-37.548,179.142,5.470,149.216
C05039=1206.939,-118.705,-37.557,179.144,5.469,149.215
C05040=1206.934,-118.456,-37.567,179.147,5.470,149.214
C05041=1206.928,-118.205,-37.576,179.149,5.470,149.214
C05042=1206.924,-117.956,-37.586,179.151,5.470,149.213
C05043=1206.918,-117.705,-37.596,179.153,5.470,149.212
C05044=1206.913,-117.456,-37.605,179.156,5.470,149.212
C05045=1206.908,-117.206,-37.614,179.158,5.470,149.211
C05046=1206.902,-116.957,-37.624,179.160,5.470,149.211
C05047=1206.897,-116.707,-37.633,179.162,5.470,149.210
C05048=1206.892,-116.457,-37.644,179.165,5.471,149.209
C05049=1206.887,-116.207,-37.652,179.167,5.470,149.209
C05050=1206.881,-115.958,-37.663,179.169,5.471,149.208
C05051=1206.876,-115.707,-37.672,179.171,5.471,149.207
C05052=1206.871,-115.458,-37.682,179.174,5.471,149.207
C05053=1206.866,-115.208,-37.691,179.176,5.471,149.206
C05054=1206.860,-114.958,-37.701,179.177,5.471,149.206
C05055=1206.855,-114.709,-37.710,179.180,5.471,149.205
C05056=1206.849,-114.459,-37.720,179.182,5.471,149.204
C05057=1206.844,-114.209,-37.729,179.185,5.471,149.203
C05058=1206.839,-113.960,-37.739,179.186,5.471,149.203
C05059=1206.834,-113.710,-37.749,179.189,5.472,149.202
C05060=1206.828,-113.460,-37.759,179.191,5.471,149.201
C05061=1206.823,-113.210,-37.769,179.193,5.472,149.201
C05062=1206.818,-112.960,-37.778,179.195,5.472,149.200
C05063=1206.813,-112.711,-37.788,179.198,5.472,149.200
C05064=1206.807,-112.461,-37.798,179.200,5.472,149.199
C05065=1206.802,-112.212,-37.807,179.202,5.473,149.198
C05066=1206.797,-111.961,-37.817,179.205,5.472,149.198
C05067=1206.792,-111.711,-37.826,179.207,5.473,149.197
C05068=1206.786,-111.462,-37.836,179.209,5.473,149.196
C05069=1206.781,-111.212,-37.847,179.211,5.473,149.196
C05070=1206.775,-110.963,-37.856,179.214,5.473,149.195
C05071=1206.770,-110.712,-37.866,179.216,5.473,149.195
C05072=1206.766,-110.463,-37.876,179.218,5.473,149.194
C05073=1206.760,-110.213,-37.885,179.221,5.473,149.193
C05074=1206.755,-109.964,-37.895,179.223,5.473,149.192
C05075=1206.749,-109.714,-37.905,179.225,5.474,149.192
C05076=1206.744,-109.463,-37.915,179.227,5.473,149.191
C05077=1206.739,-109.214,-37.925,179.230,5.474,149.190
C05078=1206.733,-108.964,-37.935,179.232,5.473,149.190
C05079=1206.728,-108.715,-37.944,179.234,5.474,149.189
C05080=1206.723,-108.465,-37.954,179.236,5.474,149.189
C05081=1206.718,-108.215,-37.964,179.239,5.474,149.188
C05082=1206.713,-107.966,-37.974,179.240,5.474,149.187
C05083=1206.707,-107.715,-37.984,179.243,5.475,149.187
C05084=1206.701,-107.466,-37.994,179.245,5.474,149.186
C05085=1206.696,-107.217,-38.003,179.248,5.475,149.185
C05086=1206.691,-106.966,-38.014,179.249,5.475,149.185
C05087=1206.686,-106.717,-38.023,179.252,5.475,149.184
C05088=1206.681,-106.467,-38.033,179.254,5.475,149.183
C05089=1206.675,-106.217,-38.043,179.257,5.475,149.183
C05090=1206.671,-105.968,-38.053,179.258,5.475,149.182
C05091=1206.665,-105.718,-38.063,179.261,5.476,149.181
C05092=1206.659,-105.468,-38.073,179.263,5.475,149.181
C05093=1206.654,-105.219,-38.083,179.266,5.476,149.180
C05094=1206.649,-104.968,-38.093,179.267,5.476,149.179
C05095=1206.644,-104.719,-38.103,179.270,5.476,149.179
C05096=1206.639,-104.470,-38.113,179.272,5.476,149.178
C05097=1206.634,-104.219,-38.123,179.274,5.476,149.178
C05098=1206.628,-103.969,-38.133,179.276,5.476,149.177
C05099=1206.623,-103.720,-38.143,179.279,5.476,149.176
C05100=1206.618,-103.470,-38.153,179.281,5.476,149.175
C05101=1206.613,-103.220,-38.163,179.283,5.477,149.175
C05102=1206.607,-102.971,-38.174,179.285,5.476,149.174
C05103=1206.602,-102.721,-38.183,179.288,5.477,149.174
C05104=1206.597,-102.470,-38.193,179.290,5.476,149.173
C05105=1206.591,-102.221,-38.203,179.292,5.477,149.172
C05106=1206.586,-101.972,-38.213,179.294,5.477,149.172
C05107=1206.581,-101.722,-38.223,179.297,5.477,149.171
C05108=1206.575,-101.451,-38.235,179.299,5.477,149.170
C05109=1206.570,-101.179,-38.246,179.302,5.477,149.169
C05110=1206.565,-100.908,-38.257,179.305,5.478,149.169
C05111=1206.558,-100.636,-38.267,179.307,5.477,149.168
C05112=1206.553,-100.386,-38.278,179.309,5.478,149.167
C05113=1206.548,-100.137,-38.287,179.311,5.478,149.167
C05114=1206.542,-99.887,-38.297,179.314,5.478,149.166
C05115=1206.537,-99.637,-38.308,179.316,5.478,149.165
C05116=1206.532,-99.388,-38.318,179.318,5.478,149.165
C05117=1206.527,-99.138,-38.328,179.320,5.478,149.164
C05118=1206.522,-98.888,-38.338,179.323,5.479,149.164
C05119=1206.516,-98.639,-38.349,179.325,5.478,149.163
C05120=1206.511,-98.389,-38.359,179.327,5.479,149.162
C05121=1206.506,-98.139,-38.369,179.330,5.478,149.161
C05122=1206.500,-97.889,-38.380,179.332,5.479,149.161
C05123=1206.495,-97.640,-38.389,179.334,5.479,149.160
C05124=1206.490,-97.390,-38.400,179.336,5.479,149.159
C05125=1206.485,-97.140,-38.410,179.339,5.479,149.159
C05126=1206.480,-96.890,-38.421,179.341,5.480,149.158
C05127=1206.474,-96.640,-38.431,179.343,5.480,149.158
C05128=1206.468,-96.391,-38.441,179.346,5.480,149.157
C05129=1206.464,-96.141,-38.451,179.348,5.480,149.156
C05130=1206.458,-95.891,-38.461,179.350,5.480,149.156
C05131=1206.453,-95.642,-38.471,179.352,5.480,149.155
C05132=1206.448,-95.392,-38.482,179.355,5.480,149.154
C05133=1206.443,-95.143,-38.493,179.357,5.480,149.154
C05134=1206.438,-94.893,-38.503,179.359,5.480,149.153
C05135=1206.432,-94.643,-38.514,179.361,5.481,149.152
C05136=1206.426,-94.393,-38.524,179.364,5.481,149.152
C05137=1206.422,-94.143,-38.534,179.366,5.481,149.151
C05138=1206.417,-93.894,-38.544,179.368,5.481,149.150
C05139=1206.412,-93.644,-38.555,179.371,5.481,149.150
C05140=1206.406,-93.394,-38.565,179.373,5.481,149.149
C05141=1206.400,-93.145,-38.575,179.375,5.481,149.148
C05142=1206.395,-92.894,-38.586,179.377,5.481,149.148
C05143=1206.390,-92.645,-38.597,179.380,5.481,149.147
C05144=1206.385,-92.395,-38.607,179.382,5.482,149.146
C05145=1206.379,-92.146,-38.617,179.384,5.482,149.146
C05146=1206.374,-91.895,-38.628,179.387,5.482,149.145
C05147=1206.369,-91.646,-38.638,179.389,5.482,149.144
C05148=1206.363,-91.396,-38.648,179.391,5.483,149.144
C05149=1206.359,-91.147,-38.660,179.393,5.482,149.143
C05150=1206.354,-90.897,-38.669,179.396,5.483,149.142
C05151=1206.349,-90.647,-38.680,179.398,5.482,149.142
C05152=1206.343,-90.398,-38.690,179.401,5.483,149.141
C05153=1206.338,-90.147,-38.701,179.402,5.483,149.140
C05154=1206.333,-89.899,-38.711,179.405,5.483,149.140
C05155=1206.328,-89.648,-38.722,179.407,5.483,149.139
C05156=1206.322,-89.399,-38.732,179.410,5.483,149.138
C05157=1206.317,-89.148,-38.743,179.412,5.483,149.138
C05158=1206.312,-88.900,-38.754,179.414,5.484,149.137
C05159=1206.306,-88.650,-38.764,179.417,5.484,149.136
C05160=1206.301,-88.400,-38.775,179.419,5.484,149.136
C05161=1206.296,-88.150,-38.785,179.422,5.484,149.135
C05162=1206.291,-87.901,-38.796,179.423,5.484,149.134
C05163=1206.285,-87.651,-38.806,179.426,5.485,149.134
C05164=1206.280,-87.401,-38.817,179.428,5.484,149.133
C05165=1206.275,-87.151,-38.827,179.431,5.485,149.132
C05166=1206.270,-86.902,-38.838,179.433,5.484,149.132
C05167=1206.265,-86.652,-38.849,179.435,5.485,149.131
C05168=1206.260,-86.402,-38.859,179.437,5.485,149.130
C05169=1206.254,-86.153,-38.870,179.440,5.485,149.130
C05170=1206.249,-85.903,-38.881,179.442,5.486,149.129
C05171=1206.243,-85.653,-38.891,179.444,5.485,149.128
C05172=1206.238,-85.403,-38.903,179.447,5.486,149.128
C05173=1206.233,-85.153,-38.913,179.449,5.486,149.127
C05174=1206.228,-84.903,-38.923,179.451,5.486,149.126
C05175=1206.223,-84.654,-38.935,179.453,5.486,149.126
C05176=1206.217,-84.404,-38.945,179.456,5.486,149.125
C05177=1206.212,-84.154,-38.956,179.458,5.486,149.125
C05178=1206.207,-83.905,-38.966,179.460,5.487,149.124
C05179=1206.202,-83.655,-38.977,179.462,5.486,149.123
C05180=1206.197,-83.406,-38.988,179.465,5.487,149.122
C05181=1206.192,-83.156,-38.999,179.468,5.487,149.122
C05182=1206.186,-82.906,-39.009,179.469,5.487,149.121
C05183=1206.181,-82.656,-39.021,179.472,5.488,149.120
C05184=1206.176,-82.406,-39.031,179.474,5.487,149.120
C05185=1206.170,-82.157,-39.042,179.477,5.488,149.119
C05186=1206.165,-81.907,-39.053,179.479,5.487,149.118
C05187=1206.160,-81.658,-39.064,179.482,5.488,149.118
C05188=1206.155,-81.408,-39.074,179.483,5.488,149.117
C05189=1206.150,-81.159,-39.085,179.486,5.488,149.116
C05190=1206.145,-80.908,-39.096,179.488,5.489,149.116
C05191=1206.139,-80.658,-39.107,179.491,5.488,149.115
C05192=1206.134,-80.409,-39.118,179.493,5.489,149.114
C05193=1206.129,-80.159,-39.128,179.495,5.489,149.114
C05194=1206.124,-79.910,-39.139,179.498,5.489,149.113
C05195=1206.119,-79.660,-39.150,179.500,5.489,149.112
C05196=1206.114,-79.410,-39.161,179.502,5.489,149.112
C05197=1206.108,-79.160,-39.172,179.505,5.490,149.111
C05198=1206.103,-78.910,-39.183,179.507,5.490,149.111
C05199=1206.097,-78.661,-39.193,179.509,5.490,149.110
C05200=1206.093,-78.411,-39.205,179.511,5.490,149.109
C05201=1206.088,-78.162,-39.216,179.514,5.490,149.108
C05202=1206.082,-77.912,-39.227,179.516,5.490,149.108
C05203=1206.077,-77.662,-39.238,179.519,5.490,149.107
C05204=1206.071,-77.413,-39.248,179.521,5.491,149.107
C05205=1206.067,-77.163,-39.260,179.523,5.491,149.106
C05206=1206.061,-76.912,-39.271,179.526,5.491,149.105
C05207=1206.056,-76.664,-39.282,179.528,5.491,149.104
C05208=1206.051,-76.414,-39.293,179.530,5.491,149.104
C05209=1206.046,-76.164,-39.304,179.532,5.491,149.103
C05210=1206.040,-75.914,-39.315,179.535,5.492,149.102
C05211=1206.035,-75.664,-39.326,179.537,5.492,149.102
C05212=1206.029,-75.394,-39.338,179.539,5.492,149.101
C05213=1206.024,-75.123,-39.349,179.542,5.492,149.100
C05214=1206.018,-74.852,-39.362,179.545,5.493,149.100
C05215=1206.012,-74.582,-39.373,179.547,5.492,149.099
C05216=1206.007,-74.332,-39.385,179.550,5.493,149.098
C05217=1206.002,-74.082,-39.397,179.552,5.493,149.098
C05218=1205.996,-73.833,-39.407,179.554,5.493,149.097
C05219=1205.991,-73.583,-39.418,179.557,5.493,149.096
C05220=1205.987,-73.334,-39.429,179.559,5.493,149.095
C05221=1205.980,-73.084,-39.440,179.561,5.494,149.095
C05222=1205.976,-72.834,-39.451,179.563,5.493,149.094
C05223=1205.971,-72.585,-39.463,179.566,5.494,149.094
C05224=1205.965,-72.334,-39.474,179.569,5.494,149.093
C05225=1205.960,-72.085,-39.485,179.571,5.494,149.092
C05226=1205.955,-71.835,-39.496,179.573,5.494,149.091
C05227=1205.950,-71.585,-39.508,179.575,5.494,149.091
C05228=1205.944,-71.336,-39.518,179.578,5.495,149.090
C05229=1205.940,-71.086,-39.530,179.580,5.495,149.089
C05230=1205.934,-70.836,-39.541,179.582,5.495,149.089
C05231=1205.929,-70.587,-39.552,179.585,5.495,149.088
C05232=1205.923,-70.337,-39.563,179.587,5.495,149.087
C05233=1205.918,-70.087,-39.575,179.589,5.496,149.087
C05234=1205.914,-69.838,-39.586,179.592,5.496,149.086
C05235=1205.908,-69.588,-39.598,179.594,5.496,149.085
C05236=1205.903,-69.338,-39.608,179.597,5.496,149.085
C05237=1205.898,-69.089,-39.619,179.599,5.496,149.084
C05238=1205.893,-68.839,-39.631,179.602,5.496,149.083
C05239=1205.887,-68.590,-39.642,179.604,5.497,149.083
C05240=1205.882,-68.340,-39.654,179.606,5.497,149.082
C05241=1205.877,-68.089,-39.665,179.608,5.497,149.081
C05242=1205.871,-67.840,-39.677,179.611,5.497,149.081
C05243=1205.866,-67.591,-39.688,179.613,5.497,149.080
C05244=1205.862,-67.341,-39.699,179.616,5.498,149.079
C05245=1205.856,-67.091,-39.711,179.618,5.498,149.079
C05246=1205.851,-66.841,-39.722,179.620,5.498,149.078
C05247=1205.845,-66.592,-39.734,179.622,5.498,149.077
C05248=1205.840,-66.342,-39.744,179.625,5.498,149.077
C05249=1205.835,-66.092,-39.756,179.628,5.499,149.076
C05250=1205.830,-65.842,-39.767,179.630,5.498,149.075
C05251=1205.824,-65.593,-39.779,179.632,5.499,149.075
C05252=1205.820,-65.344,-39.790,179.634,5.499,149.074
C05253=1205.815,-65.094,-39.801,179.637,5.499,149.073
C05254=1205.809,-64.844,-39.813,179.639,5.500,149.073
C05255=1205.805,-64.594,-39.825,179.641,5.499,149.072
C05256=1205.799,-64.345,-39.836,179.644,5.500,149.071
C05257=1205.794,-64.095,-39.847,179.646,5.499,149.071
C05258=1205.789,-63.846,-39.859,179.648,5.500,149.070
C05259=1205.784,-63.595,-39.870,179.651,5.501,149.069
C05260=1205.778,-63.345,-39.882,179.653,5.500,149.069
C05261=1205.773,-63.096,-39.893,179.656,5.501,149.068
C05262=1205.767,-62.846,-39.905,179.658,5.501,149.067
C05263=1205.763,-62.597,-39.916,179.660,5.501,149.067
C05264=1205.757,-62.347,-39.928,179.663,5.502,149.066
C05265=1205.753,-62.097,-39.939,179.665,5.501,149.065
C05266=1205.747,-61.847,-39.951,179.667,5.502,149.065
C05267=1205.742,-61.597,-39.963,179.670,5.502,149.064
C05268=1205.736,-61.349,-39.974,179.672,5.502,149.063
C05269=1205.731,-61.099,-39.986,179.675,5.502,149.063
C05270=1205.726,-60.849,-39.997,179.677,5.502,149.062
C05271=1205.721,-60.599,-40.009,179.679,5.503,149.061
C05272=1205.717,-60.350,-40.021,179.682,5.503,149.061
C05273=1205.711,-60.100,-40.033,179.684,5.503,149.060
C05274=1205.706,-59.850,-40.044,179.687,5.503,149.059
C05275=1205.700,-59.601,-40.055,179.689,5.504,149.059
C05276=1205.695,-59.351,-40.067,179.691,5.503,149.058
C05277=1205.690,-59.102,-40.079,179.694,5.504,149.057
C05278=1205.685,-58.852,-40.090,179.696,5.504,149.057
C05279=1205.680,-58.602,-40.102,179.698,5.504,149.056
C05280=1205.675,-58.352,-40.114,179.701,5.505,149.055
C05281=1205.669,-58.102,-40.126,179.703,5.504,149.055
C05282=1205.665,-57.853,-40.137,179.706,5.505,149.054
C05283=1205.659,-57.603,-40.149,179.708,5.505,149.053
C05284=1205.655,-57.354,-40.161,179.710,5.505,149.052
C05285=1205.649,-57.104,-40.172,179.713,5.506,149.052
C05286=1205.643,-56.854,-40.184,179.715,5.506,149.051
C05287=1205.639,-56.605,-40.195,179.717,5.506,149.051
C05288=1205.633,-56.355,-40.207,179.720,5.506,149.050
C05289=1205.628,-56.105,-40.219,179.722,5.506,149.049
C05290=1205.623,-55.856,-40.231,179.725,5.506,149.049
C05291=1205.618,-55.606,-40.243,179.727,5.507,149.048
C05292=1205.612,-55.356,-40.255,179.729,5.507,149.047
C05293=1205.608,-55.106,-40.266,179.732,5.507,149.047
C05294=1205.602,-54.857,-40.278,179.734,5.508,149.046
C05295=1205.597,-54.607,-40.291,179.736,5.507,149.045
C05296=1205.593,-54.358,-40.302,179.739,5.508,149.045
C05297=1205.587,-54.108,-40.314,179.742,5.508,149.044
C05298=1205.582,-53.858,-40.326,179.744,5.508,149.043
C05299=1205.577,-53.609,-40.338,179.746,5.509,149.043
C05300=1205.572,-53.359,-40.350,179.748,5.508,149.042
C05301=1205.566,-53.110,-40.361,179.751,5.509,149.041
C05302=1205.560,-52.860,-40.373,179.753,5.509,149.041
C05303=1205.556,-52.611,-40.385,179.755,5.509,149.040
C05304=1205.551,-52.361,-40.397,179.758,5.509,149.039
C05305=1205.545,-52.111,-40.409,179.761,5.510,149.038
C05306=1205.540,-51.861,-40.421,179.762,5.510,149.038
C05307=1205.535,-51.612,-40.433,179.765,5.510,149.037
C05308=1205.530,-51.362,-40.445,179.768,5.511,149.037
C05309=1205.525,-51.112,-40.457,179.770,5.510,149.036
C05310=1205.519,-50.863,-40.469,179.772,5.511,149.035
C05311=1205.515,-50.613,-40.480,179.775,5.511,149.034
C05312=1205.509,-50.363,-40.492,179.777,5.511,149.034
C05313=1205.504,-50.114,-40.505,179.779,5.512,149.033
C05314=1205.499,-49.864,-40.517,179.782,5.512,149.033
C05315=1205.494,-49.614,-40.528,179.784,5.512,149.032
C05316=1205.488,-49.344,-40.542,179.787,5.512,149.031
C05317=1205.483,-49.074,-40.555,179.790,5.513,149.030
C05318=1205.477,-48.804,-40.568,179.792,5.513,149.030
C05319=1205.472,-48.534,-40.581,179.795,5.513,149.029
C05320=1205.466,-48.284,-40.593,179.797,5.513,149.028
C05321=1205.461,-48.034,-40.605,179.800,5.514,149.028
C05322=1205.456,-47.785,-40.617,179.802,5.514,149.027
C05323=1205.451,-47.536,-40.629,179.804,5.514,149.026
C05324=1205.446,-47.286,-40.641,179.807,5.514,149.026
C05325=1205.441,-47.036,-40.653,179.809,5.514,149.025
C05326=1205.435,-46.786,-40.666,179.812,5.515,149.024
C05327=1205.430,-46.536,-40.678,179.814,5.515,149.023
C05328=1205.425,-46.287,-40.690,179.816,5.515,149.023
C05329=1205.420,-46.037,-40.701,179.819,5.516,149.022
C05330=1205.415,-45.788,-40.714,179.821,5.516,149.022
C05331=1205.410,-45.538,-40.726,179.823,5.516,149.021
C05332=1205.404,-45.289,-40.739,179.826,5.516,149.020
C05333=1205.400,-45.038,-40.751,179.829,5.517,149.019
C05334=1205.395,-44.789,-40.763,179.831,5.516,149.019
C05335=1205.389,-44.539,-40.775,179.833,5.517,149.018
C05336=1205.384,-44.290,-40.788,179.836,5.518,149.018
C05337=1205.379,-44.040,-40.800,179.838,5.518,149.017
C05338=1205.373,-43.790,-40.812,179.840,5.518,149.016
C05339=1205.369,-43.541,-40.824,179.843,5.518,149.015
C05340=1205.364,-43.291,-40.836,179.846,5.519,149.015
C05341=1205.358,-43.042,-40.848,179.848,5.518,149.014
C05342=1205.353,-42.792,-40.861,179.850,5.519,149.013
C05343=1205.348,-42.543,-40.873,179.853,5.520,149.013
C05344=1205.343,-42.292,-40.886,179.855,5.519,149.012
C05345=1205.338,-42.043,-40.898,179.857,5.520,149.011
C05346=1205.333,-41.793,-40.910,179.860,5.520,149.011
C05347=1205.327,-41.544,-40.923,179.862,5.520,149.010
C05348=1205.322,-41.294,-40.935,179.865,5.520,149.009
C05349=1205.317,-41.044,-40.947,179.867,5.521,149.009
C05350=1205.312,-40.795,-40.960,179.869,5.521,149.008
C05351=1205.306,-40.545,-40.972,179.872,5.521,149.007
C05352=1205.302,-40.295,-40.985,179.874,5.522,149.007
C05353=1205.297,-40.046,-40.997,179.876,5.521,149.006
C05354=1205.291,-39.796,-41.009,179.879,5.522,149.005
C05355=1205.286,-39.547,-41.022,179.882,5.522,149.005
C05356=1205.281,-39.297,-41.034,179.884,5.523,149.004
C05357=1205.276,-39.047,-41.046,179.887,5.522,149.003
C05358=1205.271,-38.797,-41.059,179.889,5.523,149.003
C05359=1205.266,-38.548,-41.072,179.891,5.524,149.002
C05360=1205.260,-38.298,-41.084,179.893,5.523,149.001
C05361=1205.255,-38.049,-41.096,179.896,5.524,149.001
C05362=1205.250,-37.799,-41.109,179.899,5.524,149.000
C05363=1205.245,-37.550,-41.121,179.901,5.524,148.999
C05364=1205.240,-37.299,-41.134,179.904,5.524,148.999
C05365=1205.235,-37.050,-41.146,179.906,5.525,148.998
C05366=1205.230,-36.801,-41.159,179.908,5.526,148.997
C05367=1205.225,-36.551,-41.171,179.910,5.525,148.997
C05368=1205.219,-36.302,-41.183,179.913,5.526,148.996
C05369=1205.214,-36.052,-41.197,179.916,5.526,148.995
C05370=1205.209,-35.802,-41.210,179.918,5.526,148.995
C05371=1205.204,-35.552,-41.221,179.921,5.526,148.994
C05372=1205.199,-35.303,-41.234,179.923,5.527,148.993
C05373=1205.193,-35.053,-41.247,179.926,5.527,148.993
C05374=1205.188,-34.804,-41.259,179.927,5.527,148.992
C05375=1205.184,-34.554,-41.272,179.930,5.528,148.991
C05376=1205.178,-34.304,-41.284,179.933,5.528,148.991
C05377=1205.173,-34.055,-41.297,179.935,5.528,148.990
C05378=1205.167,-33.805,-41.310,179.938,5.528,148.989
C05379=1205.163,-33.555,-41.323,179.940,5.529,148.989
C05380=1205.158,-33.306,-41.335,179.943,5.529,148.988
C05381=1205.153,-33.057,-41.348,179.945,5.529,148.987
C05382=1205.147,-32.807,-41.360,179.947,5.530,148.987
C05383=1205.143,-32.557,-41.373,179.950,5.530,148.986
C05384=1205.138,-32.307,-41.385,179.952,5.530,148.985
C05385=1205.132,-32.058,-41.399,179.954,5.531,148.985
C05386=1205.127,-31.808,-41.411,179.957,5.531,148.984
C05387=1205.122,-31.558,-41.424,179.960,5.531,148.983
C05388=1205.117,-31.309,-41.437,179.962,5.531,148.983
C05389=1205.112,-31.060,-41.449,179.964,5.532,148.982
C05390=1205.106,-30.809,-41.462,179.967,5.532,148.981
C05391=1205.101,-30.559,-41.475,179.969,5.532,148.981
C05392=1205.096,-30.310,-41.487,179.971,5.533,148.980
C05393=1205.091,-30.061,-41.500,179.974,5.533,148.979
C05394=1205.086,-29.811,-41.513,179.977,5.534,148.979
C05395=1205.080,-29.561,-41.526,179.979,5.533,148.978
C05396=1205.075,-29.312,-41.539,179.982,5.534,148.977
C05397=1205.070,-29.062,-41.551,179.984,5.535,148.977
C05398=1205.066,-28.812,-41.564,179.986,5.535,148.976
C05399=1205.061,-28.563,-41.577,179.988,5.535,148.975
C05400=1205.055,-28.313,-41.590,179.991,5.535,148.975
C05401=1205.050,-28.063,-41.603,179.994,5.536,148.974
C05402=1205.045,-27.814,-41.616,179.996,5.536,148.973
C05403=1205.040,-27.565,-41.628,179.998,5.536,148.973
C05404=1205.035,-27.315,-41.642,-179.999,5.536,148.972
C05405=1205.030,-27.065,-41.655,-179.997,5.537,148.971
C05406=1205.024,-26.816,-41.667,-179.995,5.537,148.971
C05407=1205.019,-26.566,-41.681,-179.992,5.537,148.970
C05408=1205.014,-26.316,-41.693,-179.989,5.538,148.969
C05409=1205.009,-26.067,-41.706,-179.987,5.538,148.969
C05410=1205.004,-25.817,-41.719,-179.985,5.538,148.968
C05411=1204.999,-25.568,-41.733,-179.982,5.538,148.967
C05412=1204.994,-25.319,-41.745,-179.979,5.539,148.966
C05413=1204.989,-25.069,-41.758,-179.977,5.540,148.966
C05414=1204.983,-24.819,-41.772,-179.975,5.539,148.965
C05415=1204.979,-24.569,-41.785,-179.972,5.540,148.965
C05416=1204.974,-24.320,-41.797,-179.970,5.540,148.964
C05417=1204.968,-24.070,-41.810,-179.967,5.541,148.963
C05418=1204.963,-23.820,-41.823,-179.965,5.540,148.963
C05419=1204.958,-23.571,-41.836,-179.962,5.541,148.962
C05420=1204.953,-23.301,-41.851,-179.960,5.541,148.961
C05421=1204.947,-23.032,-41.864,-179.957,5.542,148.960
C05422=1204.941,-22.762,-41.878,-179.954,5.542,148.960
C05423=1204.936,-22.493,-41.893,-179.952,5.543,148.959
C05424=1204.931,-22.243,-41.906,-179.949,5.543,148.958
C05425=1204.926,-21.993,-41.919,-179.947,5.543,148.958
C05426=1204.920,-21.744,-41.932,-179.944,5.543,148.957
C05427=1204.915,-21.494,-41.945,-179.942,5.544,148.956
C05428=1204.910,-21.245,-41.959,-179.939,5.545,148.956
C05429=1204.905,-20.995,-41.972,-179.937,5.544,148.955
C05430=1204.901,-20.745,-41.985,-179.935,5.545,148.954
C05431=1204.895,-20.496,-41.998,-179.932,5.545,148.954
C05432=1204.890,-20.246,-42.011,-179.929,5.546,148.953
C05433=1204.885,-19.997,-42.025,-179.927,5.546,148.952
C05434=1204.880,-19.747,-42.037,-179.925,5.546,148.952
C05435=1204.874,-19.497,-42.051,-179.922,5.547,148.951
C05436=1204.869,-19.248,-42.063,-179.920,5.547,148.950
C05437=1204.865,-18.998,-42.077,-179.917,5.548,148.950
C05438=1204.859,-18.749,-42.090,-179.915,5.548,148.949
C05439=1204.855,-18.499,-42.103,-179.912,5.548,148.948
C05440=1204.849,-18.250,-42.117,-179.910,5.548,148.948
C05441=1204.844,-18.000,-42.130,-179.907,5.549,148.947
C05442=1204.839,-17.750,-42.143,-179.905,5.549,148.946
C05443=1204.834,-17.501,-42.157,-179.902,5.549,148.946
C05444=1204.829,-17.251,-42.170,-179.900,5.550,148.945
C05445=1204.824,-17.002,-42.183,-179.897,5.550,148.944
C05446=1204.819,-16.752,-42.197,-179.895,5.551,148.944
C05447=1204.813,-16.503,-42.210,-179.893,5.551,148.943
C05448=1204.808,-16.252,-42.223,-179.890,5.551,148.942
C05449=1204.803,-16.004,-42.237,-179.887,5.552,148.942
C05450=1204.798,-15.753,-42.250,-179.885,5.552,148.941
C05451=1204.793,-15.504,-42.263,-179.883,5.552,148.941
C05452=1204.788,-15.254,-42.277,-179.881,5.553,148.940
C05453=1204.783,-15.005,-42.290,-179.878,5.553,148.939
C05454=1204.778,-14.755,-42.304,-179.875,5.554,148.938
C05455=1204.772,-14.506,-42.317,-179.873,5.554,148.938
C05456=1204.768,-14.256,-42.330,-179.870,5.554,148.937
C05457=1204.762,-14.007,-42.344,-179.868,5.554,148.936
C05458=1204.757,-13.757,-42.357,-179.865,5.555,148.936
C05459=1204.752,-13.508,-42.371,-179.863,5.556,148.935
C05460=1204.747,-13.258,-42.384,-179.860,5.556,148.935
C05461=1204.742,-13.009,-42.398,-179.858,5.556,148.934
C05462=1204.737,-12.758,-42.411,-179.856,5.556,148.933
C05463=1204.732,-12.509,-42.425,-179.853,5.557,148.932
C05464=1204.726,-12.259,-42.438,-179.850,5.557,148.932
C05465=1204.722,-12.010,-42.452,-179.848,5.558,148.931
C05466=1204.716,-11.760,-42.465,-179.846,5.558,148.931
C05467=1204.711,-11.510,-42.479,-179.843,5.558,148.930
C05468=1204.706,-11.261,-42.492,-179.841,5.559,148.929
C05469=1204.701,-11.011,-42.506,-179.838,5.559,148.928
C05470=1204.696,-10.762,-42.519,-179.835,5.560,148.928
C05471=1204.691,-10.512,-42.533,-179.833,5.559,148.927
C05472=1204.686,-10.262,-42.547,-179.831,5.560,148.926
C05473=1204.681,-10.013,-42.560,-179.828,5.560,148.926
C05474=1204.676,-9.763,-42.574,-179.826,5.561,148.925
C05475=1204.670,-9.514,-42.587,-179.823,5.562,148.925
C05476=1204.666,-9.265,-42.601,-179.821,5.561,148.924
C05477=1204.661,-9.014,-42.615,-179.818,5.562,148.923
C05478=1204.655,-8.765,-42.629,-179.816,5.562,148.922
C05479=1204.651,-8.515,-42.642,-179.813,5.563,148.922
C05480=1204.645,-8.266,-42.656,-179.811,5.563,148.921
C05481=1204.640,-8.017,-42.670,-179.808,5.564,148.921
C05482=1204.636,-7.767,-42.683,-179.806,5.564,148.920
C05483=1204.630,-7.518,-42.697,-179.804,5.564,148.919
C05484=1204.625,-7.268,-42.711,-179.801,5.565,148.919
C05485=1204.620,-7.019,-42.724,-179.798,5.565,148.918
C05486=1204.615,-6.769,-42.738,-179.796,5.566,148.917
C05487=1204.610,-6.519,-42.752,-179.794,5.566,148.917
